messageStringBuilder(
	sFormat := message,
	arg1 := THIS^.AnyToArg(currentValueAsString),
	arg2 := THIS^.AnyToArg(minimumValueAsString)
);

THIS^.assertorContainer.assertor.assert.dateAndTime.simple.dateAndTime.valueIsMin(
	currentValue	:= valueToTest,
	minimumValue	:= minimumValue,
	message			:= ''
);

THIS^.AssertEquals_BOOL(
	Expected 	:= assertionIsWrong,
	Actual 		:= THIS^.assertorContainer.wasAssertionWrong,
	Message 	:= messageStringBuilder.sOut
);
END_METHOD

(*

short summary
==================
This test method tests ``assert.dateAndTime.simple.dateAndTime.valueIsNotEqualTo``
method of CNM_AssertionInterfaces library, 
it provides the possibility to handover test data via parameter 


.. <legal notes>

legal notes
=================
| SPDX-FileCopyrightText: © 2022 ekvip automation GmbH <info@ekvip.de>
| SPDX-License-Identifier: Apache-2.0
| For details check: Apache-2.0_

.. _Apache-2.0: https://www.apache.org/licenses/LICENSE-2.0

.. </legal notes>

parameters
==========

*)

METHOD testValueIsNotEqualTo 
VAR_INPUT
	(* for the test it's the parameter ``currentValue`` *)
	valueToTest		:DT;
	(* for the test it's the parameter ``unexpectedValue`` *)
	unexpectedValue	:DT;
END_VAR
VAR
	(* just the expectation if the assertion to test must be worng or true *)
	assertionIsWrong		:BOOL;
	(* contains the format string for the test message *)
	message					:Tc2_System.T_MaxString;
	(* TwinCAT printf with the test message *)
	messageStringBuilder	:Tc2_Utilities.FB_FormatString;
	(* dt value of ``currentValue`` as string *)
	currentValueAsString	:STRING(22);
	(* dt value of ``unexpectedValue`` as string *)
	unexpectedValueAsString	:STRING(22);
END_VAR
THIS^.assertorContainer.resetAssertor();

assertionIsWrong := (valueToTest = unexpectedValue);
message := SEL(
	assertionIsWrong,
	'currentValue is %s expectedValue is %s assertion must be TRUE', 
	'currentValue is %s expectedValue is %s assertion must be FALSE'
);
currentValueAsString := TO_STRING(valueToTest);
unexpectedValueAsString := TO_STRING(unexpectedValue);

messageStringBuilder(
	sFormat := message,
	arg1 := THIS^.AnyToArg(currentValueAsString),
	arg2 := THIS^.AnyToArg(unexpectedValueAsString)
);

THIS^.assertorContainer.assertor.assert.dateAndTime.simple.dateAndTime.valueIsNotEqualTo(
	currentValue	:= valueToTest,
	unexpectedValue	:= unexpectedValue,
	message			:= ''
);

THIS^.AssertEquals_BOOL(
	Expected 	:= assertionIsWrong,
	Actual 		:= THIS^.assertorContainer.wasAssertionWrong,
	Message 	:= messageStringBuilder.sOut
);
END_METHOD

END_FUNCTION_BLOCK

// ---- AssertionTester/AssertionTests/DateTimeAssertions/classes/DateAssertionTests.TcPOU
(*

short summary
==================
This class tests all methods of DATE assertions
with various combinations of inputs and checks expected 
outputs are satisfied or not

.. <legal notes>

legal notes
=================
| SPDX-FileCopyrightText: © 2022 ekvip automation GmbH <info@ekvip.de>
| SPDX-License-Identifier: Apache-2.0
| For details check: Apache-2.0_

.. _Apache-2.0: https://www.apache.org/licenses/LICENSE-2.0

.. </legal notes>

methods and properties
======================

*)


FUNCTION_BLOCK DateAssertionTests EXTENDS AbstractAssertorTest
VAR
	
END_VAR
VAR CONSTANT
	(* prefix to unify the test names *)
	TEST_NAME_PREFIX		:STRING := 'assert.dateAndTime.simple.dateOnly.';
	(* max value of a DWORD *)
	{attribute 'hide'}
	MAX_DWORD				:DWORD := 16#FFFF_FFFF;
	(* min value of a DWORD *)
	{attribute 'hide'}
	MIN_DWORD				:DWORD := 16#0000_0000;
	(* only the msb is set *)
	{attribute 'hide'}
	MSB_ONLY				:DWORD := 16#8000_0000;
	(* only the msb is set *)
	{attribute 'hide'}
	LSB_ONLY				:DWORD := 16#0000_0001;
	(* all bits set except the msb *)
	{attribute 'hide'}
	WITHOUT_MSB 			:DWORD := 16#7FFF_FFFF;
	(* for every nibble is the msb set only *)
	{attribute 'hide'}
	ALL_NIBBLE_MSB			:DWORD := 16#8888_8888;
	(* for every nibble is the msb unset only *)
	{attribute 'hide'}
	WITHOUT_NIBBLE_MSB		:DWORD := 16#7777_7777;
	(* for every nibble is the lsb set only *)
	{attribute 'hide'}
	ALL_NIBBLE_LSB			:DWORD := 16#1111_1111;
	(* every bit is set except the lsb *)
	{attribute 'hide'}
	LSB_IS_UNSET			:DWORD := 16#FFFF_FFFE;
	(* max vale of date and time *)
	DATE_MAX				:DATE := TO_DATE(MAX_DWORD);
	(* min vale of date and time *)
	DATE_MIN				:DATE := TO_DATE(MIN_DWORD);
	(* only the msb is set *)
	DATE_MSB_ONLY			:DATE := TO_DATE(MSB_ONLY);
	(* all bits set except the msb *)
	DATE_WITHOUT_MSB 		:DATE := TO_DATE(WITHOUT_MSB);
	(* for every nibble is the msb set only *)
	DATE_ALL_NIBBLE_MSB		:DATE := TO_DATE(ALL_NIBBLE_MSB);
	(* for every nibble is the msb unset only *)
	DATE_WITHOUT_NIBBLE_MSB	:DATE := TO_DATE(WITHOUT_NIBBLE_MSB);
	(* for every nibble is the lsb set only *)
	DATE_ALL_NIBBLE_LSB		:DATE := TO_DATE(ALL_NIBBLE_LSB);	
	(* every bit is set except the lsb *)
	DATE_LSB_IS_UNSET		:DATE := TO_DATE(LSB_IS_UNSET);
	(* only the msb is set *)
	DATE_LSB_ONLY			:DATE := TO_DATE(LSB_ONLY);
END_VAR

THIS^.runValueIsEqualToTests();
THIS^.runValueIsGreaterThanTests();
THIS^.runValueIsInRangeOfTests();
THIS^.runValueIsLessThanTests();
THIS^.runValueIsMaxTests();
THIS^.runValueIsMinTests();
THIS^.runValueIsNotEqualToTests();

(*

short summary
==================
This test method is a helper function to create a unified test name

.. <legal notes>

legal notes
=================
| SPDX-FileCopyrightText: © 2022 ekvip automation GmbH <info@ekvip.de>
| SPDX-License-Identifier: Apache-2.0
| For details check: Apache-2.0_

.. _Apache-2.0: https://www.apache.org/licenses/LICENSE-2.0

.. </legal notes>

parameters
==========

*)

METHOD PROTECTED getTestNameFor :Tc2_System.T_MaxString
VAR_INPUT
	(* name of the method to test, to create a unified test name *)
	nameOfMethodToTest	:Tc2_System.T_MaxString;
END_VAR
getTestNameFor := Tc2_Standard.CONCAT(THIS^.TEST_NAME_PREFIX, nameOfMethodToTest);
END_METHOD

(*

short summary
==================
This test method tests ``assert.dateAndTime.simple.dateOnly.valueIsEqualTo``
method of CNM_AssertionInterfaces library with various inputs

.. <legal notes>

legal notes
=================
| SPDX-FileCopyrightText: © 2022 ekvip automation GmbH <info@ekvip.de>
| SPDX-License-Identifier: Apache-2.0
| For details check: Apache-2.0_

.. _Apache-2.0: https://www.apache.org/licenses/LICENSE-2.0

.. </legal notes>

*)

METHOD runValueIsEqualToTests
RETURN (NOT TcUnit.TEST_ORDERED(THIS^.getTestNameFor('valueIsEqualTo')));

THIS^.testValueIsEqualTo(
	valueToTest := THIS^.DATE_MAX,
	expected := THIS^.DATE_MAX
);
THIS^.testValueIsEqualTo(
	valueToTest := THIS^.DATE_MIN,
	expected := THIS^.DATE_MIN
);
THIS^.testValueIsEqualTo(
	valueToTest := THIS^.DATE_MIN,
	expected := THIS^.DATE_MAX
);
THIS^.testValueIsEqualTo(
	valueToTest := THIS^.DATE_MAX,
	expected := THIS^.DATE_MIN
);
THIS^.testValueIsEqualTo(
	valueToTest := THIS^.DATE_ALL_NIBBLE_LSB,
	expected := THIS^.DATE_ALL_NIBBLE_LSB
);
THIS^.testValueIsEqualTo(
	valueToTest := THIS^.DATE_LSB_ONLY,
	expected := THIS^.DATE_MSB_ONLY
);
THIS^.testValueIsEqualTo(
	valueToTest := THIS^.DATE_MSB_ONLY,
	expected := THIS^.DATE_MSB_ONLY
);
THIS^.testValueIsEqualTo(
	valueToTest := THIS^.DATE_MSB_ONLY,
	expected := THIS^.DATE_LSB_ONLY
);

TcUnit.TEST_FINISHED();
END_METHOD

(*

short summary
==================
This test method tests ``assert.dateAndTime.simple.dateOnly.valueIsGreaterThan``
method of CNM_AssertionInterfaces library with various inputs

.. <legal notes>

legal notes
=================
| SPDX-FileCopyrightText: © 2022 ekvip automation GmbH <info@ekvip.de>
| SPDX-License-Identifier: Apache-2.0
| For details check: Apache-2.0_

.. _Apache-2.0: https://www.apache.org/licenses/LICENSE-2.0

.. </legal notes>

*)

METHOD runValueIsGreaterThanTests
RETURN (NOT TcUnit.TEST_ORDERED(THIS^.getTestNameFor('valueIsGreaterThan')));

THIS^.testValueIsGreaterThan(
	valueToTest := THIS^.DATE_MAX,
	lessValue := THIS^.DATE_MAX
);
THIS^.testValueIsGreaterThan(
	valueToTest := THIS^.DATE_MIN,
	lessValue := THIS^.DATE_MIN
);
THIS^.testValueIsGreaterThan(
	valueToTest := THIS^.DATE_MIN,
	lessValue := THIS^.DATE_MAX
);
THIS^.testValueIsGreaterThan(
	valueToTest := THIS^.DATE_MAX,
	lessValue := THIS^.DATE_MIN
);
THIS^.testValueIsGreaterThan(
	valueToTest := THIS^.DATE_ALL_NIBBLE_LSB,
	lessValue := THIS^.DATE_ALL_NIBBLE_LSB
);
THIS^.testValueIsGreaterThan(
	valueToTest := THIS^.DATE_ALL_NIBBLE_MSB,
	lessValue := THIS^.DATE_ALL_NIBBLE_LSB
);
THIS^.testValueIsGreaterThan(
	valueToTest := THIS^.DATE_ALL_NIBBLE_LSB,
	lessValue := THIS^.DATE_ALL_NIBBLE_MSB
);
THIS^.testValueIsGreaterThan(
	valueToTest := THIS^.DATE_LSB_ONLY,
	lessValue := THIS^.DATE_MSB_ONLY
);
THIS^.testValueIsGreaterThan(
	valueToTest := THIS^.DATE_MSB_ONLY,
	lessValue := THIS^.DATE_MSB_ONLY
);
THIS^.testValueIsGreaterThan(
	valueToTest := THIS^.DATE_MSB_ONLY,
	lessValue := THIS^.DATE_LSB_ONLY
);
THIS^.testValueIsGreaterThan(
	valueToTest := THIS^.DATE_LSB_IS_UNSET,
	lessValue := THIS^.DATE_MAX
);
THIS^.testValueIsGreaterThan(
	valueToTest := THIS^.DATE_MAX,
	lessValue := THIS^.DATE_LSB_IS_UNSET
);
TcUnit.TEST_FINISHED();
END_METHOD

(*

short summary
==================
This test method tests ``assert.dateAndTime.simple.dateOnly.valueIsInRangeOf``
method of CNM_AssertionInterfaces library with various inputs

.. <legal notes>

legal notes
=================
| SPDX-FileCopyrightText: © 2022 ekvip automation GmbH <info@ekvip.de>
| SPDX-License-Identifier: Apache-2.0
| For details check: Apache-2.0_

.. _Apache-2.0: https://www.apache.org/licenses/LICENSE-2.0

.. </legal notes>

*)

METHOD runValueIsInRangeOfTests
RETURN (NOT TcUnit.TEST_ORDERED(THIS^.getTestNameFor('valueIsInRangeOf')));

THIS^.testValueIsInRangeOf(
	lowerLimit := THIS^.DATE_MIN,
	valueToTest := THIS^.DATE_MAX,
	upperLimit	:= THIS^.DATE_MAX
);
THIS^.testValueIsInRangeOf(
	lowerLimit := THIS^.DATE_MIN,
	valueToTest := THIS^.DATE_MIN,
	upperLimit	:= THIS^.DATE_MAX
);
THIS^.testValueIsInRangeOf(
	lowerLimit := THIS^.DATE_MAX,
	valueToTest := THIS^.DATE_MAX,
	upperLimit	:= THIS^.DATE_MIN
);
THIS^.testValueIsInRangeOf(
	lowerLimit := THIS^.DATE_MAX,
	valueToTest := THIS^.DATE_MIN,
	upperLimit	:= THIS^.DATE_MIN
);
THIS^.testValueIsInRangeOf(
	lowerLimit := THIS^.DATE_LSB_IS_UNSET,
	valueToTest := THIS^.DATE_MIN,
	upperLimit	:= THIS^.DATE_MAX
);
THIS^.testValueIsInRangeOf(
	lowerLimit := THIS^.DATE_MIN,
	valueToTest := THIS^.DATE_LSB_IS_UNSET,
	upperLimit	:= THIS^.DATE_MAX
);
THIS^.testValueIsInRangeOf(
	lowerLimit := THIS^.DATE_LSB_IS_UNSET,
	valueToTest := THIS^.DATE_LSB_IS_UNSET,
	upperLimit	:= THIS^.DATE_LSB_IS_UNSET
);
THIS^.testValueIsInRangeOf(
	lowerLimit := THIS^.DATE_ALL_NIBBLE_LSB,
	valueToTest := THIS^.DATE_LSB_IS_UNSET,
	upperLimit	:= THIS^.DATE_ALL_NIBBLE_MSB
);
THIS^.testValueIsInRangeOf(
	lowerLimit := THIS^.DATE_LSB_IS_UNSET,
	valueToTest := THIS^.DATE_ALL_NIBBLE_LSB,
	upperLimit	:= THIS^.DATE_ALL_NIBBLE_MSB
);
THIS^.testValueIsInRangeOf(
	lowerLimit := THIS^.DATE_LSB_ONLY,
	valueToTest := THIS^.DATE_WITHOUT_MSB,
	upperLimit	:= THIS^.DATE_MSB_ONLY
);
THIS^.testValueIsInRangeOf(
	lowerLimit := THIS^.DATE_WITHOUT_MSB,
	valueToTest := THIS^.DATE_LSB_ONLY,
	upperLimit	:= THIS^.DATE_MSB_ONLY
);
THIS^.testValueIsInRangeOf(
	lowerLimit := THIS^.DATE_WITHOUT_NIBBLE_MSB,
	valueToTest := THIS^.DATE_MAX,
	upperLimit	:= THIS^.DATE_ALL_NIBBLE_MSB
);
THIS^.testValueIsInRangeOf(
	lowerLimit := THIS^.DATE_WITHOUT_NIBBLE_MSB,
	valueToTest := THIS^.DATE_MIN,
	upperLimit	:= THIS^.DATE_ALL_NIBBLE_MSB
);
THIS^.testValueIsInRangeOf(
	lowerLimit := THIS^.DATE_WITHOUT_NIBBLE_MSB,
	valueToTest := THIS^.DATE_WITHOUT_NIBBLE_MSB,
	upperLimit	:= THIS^.DATE_ALL_NIBBLE_MSB
);
THIS^.testValueIsInRangeOf(
	lowerLimit := THIS^.DATE_WITHOUT_NIBBLE_MSB,
	valueToTest := THIS^.DATE_ALL_NIBBLE_MSB,
	upperLimit	:= THIS^.DATE_ALL_NIBBLE_MSB
);
TcUnit.TEST_FINISHED();
END_METHOD

(*

short summary
==================
This test method tests ``assert.dateAndTime.simple.dateOnly.valueIsLessThan``
method of CNM_AssertionInterfaces library with various inputs

.. <legal notes>

legal notes
=================
| SPDX-FileCopyrightText: © 2022 ekvip automation GmbH <info@ekvip.de>
| SPDX-License-Identifier: Apache-2.0
| For details check: Apache-2.0_

.. _Apache-2.0: https://www.apache.org/licenses/LICENSE-2.0

.. </legal notes>

*)

METHOD runValueIsLessThanTests
RETURN (NOT TcUnit.TEST_ORDERED(THIS^.getTestNameFor('valueIsLessThan')));

THIS^.testValueIsLessThan(
	valueToTest := THIS^.DATE_MAX,
	greaterValue := THIS^.DATE_MAX
);
THIS^.testValueIsLessThan(
	valueToTest := THIS^.DATE_MIN,
	greaterValue := THIS^.DATE_MIN
);
THIS^.testValueIsLessThan(
	valueToTest := THIS^.DATE_MIN,
	greaterValue := THIS^.DATE_MAX
);
THIS^.testValueIsLessThan(
	valueToTest := THIS^.DATE_MAX,
	greaterValue := THIS^.DATE_MIN
);
THIS^.testValueIsLessThan(
	valueToTest := THIS^.DATE_ALL_NIBBLE_LSB,
	greaterValue := THIS^.DATE_ALL_NIBBLE_LSB
);
THIS^.testValueIsLessThan(
	valueToTest := THIS^.DATE_ALL_NIBBLE_MSB,
	greaterValue := THIS^.DATE_ALL_NIBBLE_LSB
);
THIS^.testValueIsLessThan(
	valueToTest := THIS^.DATE_ALL_NIBBLE_LSB,
	greaterValue := THIS^.DATE_ALL_NIBBLE_MSB
);
THIS^.testValueIsLessThan(
	valueToTest := THIS^.DATE_LSB_ONLY,
	greaterValue := THIS^.DATE_MSB_ONLY
);
THIS^.testValueIsLessThan(
	valueToTest := THIS^.DATE_MSB_ONLY,
	greaterValue := THIS^.DATE_MSB_ONLY
);
THIS^.testValueIsLessThan(
	valueToTest := THIS^.DATE_MSB_ONLY,
	greaterValue := THIS^.DATE_LSB_ONLY
);
THIS^.testValueIsLessThan(
	valueToTest := THIS^.DATE_LSB_IS_UNSET,
	greaterValue := THIS^.DATE_MAX
);
THIS^.testValueIsLessThan(
	valueToTest := THIS^.DATE_MAX,
	greaterValue := THIS^.DATE_LSB_IS_UNSET
);
TcUnit.TEST_FINISHED();
END_METHOD

(*

short summary
==================
This test method tests ``assert.dateAndTime.simple.dateOnly.valueIsMax``
method of CNM_AssertionInterfaces library with various inputs

.. <legal notes>

legal notes
=================
| SPDX-FileCopyrightText: © 2022 ekvip automation GmbH <info@ekvip.de>
| SPDX-License-Identifier: Apache-2.0
| For details check: Apache-2.0_

.. _Apache-2.0: https://www.apache.org/licenses/LICENSE-2.0

.. </legal notes>

*)

METHOD runValueIsMaxTests
RETURN (NOT TcUnit.TEST_ORDERED(THIS^.getTestNameFor('valueIsMax')));

THIS^.testValueIsMax(
	valueToTest := THIS^.DATE_MAX,
	maximumValue := THIS^.DATE_MAX
);
THIS^.testValueIsMax(
	valueToTest := THIS^.DATE_MIN,
	maximumValue := THIS^.DATE_MIN
);
THIS^.testValueIsMax(
	valueToTest := THIS^.DATE_MIN,
	maximumValue := THIS^.DATE_MAX
);
THIS^.testValueIsMax(
	valueToTest := THIS^.DATE_MAX,
	maximumValue := THIS^.DATE_MIN
);
THIS^.testValueIsMax(
	valueToTest := THIS^.DATE_ALL_NIBBLE_LSB,
	maximumValue := THIS^.DATE_ALL_NIBBLE_LSB
);
THIS^.testValueIsMax(
	valueToTest := THIS^.DATE_ALL_NIBBLE_MSB,
	maximumValue := THIS^.DATE_ALL_NIBBLE_LSB
);
THIS^.testValueIsMax(
	valueToTest := THIS^.DATE_ALL_NIBBLE_LSB,
	maximumValue := THIS^.DATE_ALL_NIBBLE_MSB
);
THIS^.testValueIsMax(
	valueToTest := THIS^.DATE_LSB_ONLY,
	maximumValue := THIS^.DATE_MSB_ONLY
);
THIS^.testValueIsMax(
	valueToTest := THIS^.DATE_MSB_ONLY,
	maximumValue := THIS^.DATE_MSB_ONLY
);
THIS^.testValueIsMax(
	valueToTest := THIS^.DATE_MSB_ONLY,
	maximumValue := THIS^.DATE_LSB_ONLY
);
THIS^.testValueIsMax(
	valueToTest := THIS^.DATE_LSB_IS_UNSET,
	maximumValue := THIS^.DATE_MAX
);
THIS^.testValueIsMax(
	valueToTest := THIS^.DATE_MAX,
	maximumValue := THIS^.DATE_LSB_IS_UNSET
);
TcUnit.TEST_FINISHED();
END_METHOD

(*

short summary
==================
This test method tests ``assert.dateAndTime.simple.dateOnly.valueIsMin``
method of CNM_AssertionInterfaces library with various inputs

.. <legal notes>

legal notes
=================
| SPDX-FileCopyrightText: © 2022 ekvip automation GmbH <info@ekvip.de>
| SPDX-License-Identifier: Apache-2.0
| For details check: Apache-2.0_

.. _Apache-2.0: https://www.apache.org/licenses/LICENSE-2.0

.. </legal notes>

*)

METHOD runValueIsMinTests
RETURN (NOT TcUnit.TEST_ORDERED(THIS^.getTestNameFor('valueIsMin')));

THIS^.testValueIsMin(
	valueToTest := THIS^.DATE_MAX,
	minimumValue := THIS^.DATE_MAX
);
THIS^.testValueIsMin(
	valueToTest := THIS^.DATE_MIN,
	minimumValue := THIS^.DATE_MIN
);
THIS^.testValueIsMin(
	valueToTest := THIS^.DATE_MIN,
	minimumValue := THIS^.DATE_MAX
);
THIS^.testValueIsMin(
	valueToTest := THIS^.DATE_MAX,
	minimumValue := THIS^.DATE_MIN
);
THIS^.testValueIsMin(
	valueToTest := THIS^.DATE_ALL_NIBBLE_LSB,
	minimumValue := THIS^.DATE_ALL_NIBBLE_LSB
);
THIS^.testValueIsMin(
	valueToTest := THIS^.DATE_ALL_NIBBLE_MSB,
	minimumValue := THIS^.DATE_ALL_NIBBLE_LSB
);
THIS^.testValueIsMin(
	valueToTest := THIS^.DATE_ALL_NIBBLE_LSB,
	minimumValue := THIS^.DATE_ALL_NIBBLE_MSB
);
THIS^.testValueIsMin(
	valueToTest := THIS^.DATE_LSB_ONLY,
	minimumValue := THIS^.DATE_MSB_ONLY
);
THIS^.testValueIsMin(
	valueToTest := THIS^.DATE_MSB_ONLY,
	minimumValue := THIS^.DATE_MSB_ONLY
);
THIS^.testValueIsMin(
	valueToTest := THIS^.DATE_MSB_ONLY,
	minimumValue := THIS^.DATE_LSB_ONLY
);
THIS^.testValueIsMin(
	valueToTest := THIS^.DATE_LSB_IS_UNSET,
	minimumValue := THIS^.DATE_MAX
);
THIS^.testValueIsMin(
	valueToTest := THIS^.DATE_MAX,
	minimumValue := THIS^.DATE_LSB_IS_UNSET
);
TcUnit.TEST_FINISHED();
END_METHOD

(*

short summary
==================
This test method tests ``assert.dateAndTime.simple.dateOnly.valueIsNotEqualTo``
method of CNM_AssertionInterfaces library with various inputs

.. <legal notes>

legal notes
=================
| SPDX-FileCopyrightText: © 2022 ekvip automation GmbH <info@ekvip.de>
| SPDX-License-Identifier: Apache-2.0
| For details check: Apache-2.0_

.. _Apache-2.0: https://www.apache.org/licenses/LICENSE-2.0

.. </legal notes>

*)

METHOD runValueIsNotEqualToTests
RETURN (NOT TcUnit.TEST_ORDERED(THIS^.getTestNameFor('valueIsNotEqualTo')));

THIS^.testValueIsNotEqualTo(
	valueToTest := THIS^.DATE_MAX,
	unexpectedValue := THIS^.DATE_MAX
);
THIS^.testValueIsNotEqualTo(
	valueToTest := THIS^.DATE_MIN,
	unexpectedValue := THIS^.DATE_MIN
);
THIS^.testValueIsNotEqualTo(
	valueToTest := THIS^.DATE_MIN,
	unexpectedValue := THIS^.DATE_MAX
);
THIS^.testValueIsNotEqualTo(
	valueToTest := THIS^.DATE_MAX,
	unexpectedValue := THIS^.DATE_MIN
);
THIS^.testValueIsNotEqualTo(
	valueToTest := THIS^.DATE_ALL_NIBBLE_LSB,
	unexpectedValue := THIS^.DATE_ALL_NIBBLE_LSB
);
THIS^.testValueIsNotEqualTo(
	valueToTest := THIS^.DATE_LSB_ONLY,
	unexpectedValue := THIS^.DATE_MSB_ONLY
);
THIS^.testValueIsNotEqualTo(
	valueToTest := THIS^.DATE_MSB_ONLY,
	unexpectedValue := THIS^.DATE_MSB_ONLY
);
THIS^.testValueIsNotEqualTo(
	valueToTest := THIS^.DATE_MSB_ONLY,
	unexpectedValue := THIS^.DATE_LSB_ONLY
);

TcUnit.TEST_FINISHED();
END_METHOD

(*

short summary
==================
This test method tests ``assert.dateAndTime.simple.dateOnly.valueIsEqualTo``
method of CNM_AssertionInterfaces library, 
it provides the possibility to handover test data via parameter 


.. <legal notes>

legal notes
=================
| SPDX-FileCopyrightText: © 2022 ekvip automation GmbH <info@ekvip.de>
| SPDX-License-Identifier: Apache-2.0
| For details check: Apache-2.0_

.. _Apache-2.0: https://www.apache.org/licenses/LICENSE-2.0

.. </legal notes>

parameters
==========

*)

METHOD testValueIsEqualTo 
VAR_INPUT
	(* for the test it's the parameter ``currentValue`` *)
	valueToTest	:DATE;
	(* for the test it's the parameter ``expectedValue`` *)
	expected	:DATE;
END_VAR
VAR
	(* just the expectation if the assertion to test must be worng or true *)
	assertionIsWrong		:BOOL;
	(* contains the format string for the test message *)
	message					:Tc2_System.T_MaxString;
	(* TwinCAT printf with the test message *)
	messageStringBuilder	:Tc2_Utilities.FB_FormatString;
	(* DATE value of ``currentValue`` as string *)
	currentValueAsString	:STRING(22);
	(* DATE value of ``expectedValue`` as string *)
	expectedValueAsString	:STRING(22);
END_VAR
THIS^.assertorContainer.resetAssertor();

assertionIsWrong := (valueToTest <> expected);
message := SEL(
	assertionIsWrong,
	'currentValue is %s expectedValue is %s assertion must be TRUE', 
	'currentValue is %s expectedValue is %s assertion must be FALSE'
);
currentValueAsString := TO_STRING(valueToTest);
expectedValueAsString := TO_STRING(expected);

messageStringBuilder(
	sFormat := message,
	arg1 := THIS^.AnyToArg(currentValueAsString),
	arg2 := THIS^.AnyToArg(expectedValueAsString)
);

THIS^.assertorContainer.assertor.assert.dateAndTime.simple.dateOnly.valueIsEqualTo(
	currentValue	:= valueToTest,
	expectedValue	:= expected,
	message			:= ''
);

THIS^.AssertEquals_BOOL(
	Expected 	:= assertionIsWrong,
	Actual 		:= THIS^.assertorContainer.wasAssertionWrong,
	Message 	:= messageStringBuilder.sOut
);
END_METHOD

(*

short summary
==================
This test method tests ``assert.dateAndTime.simple.dateOnly.valueIsGreaterThan``
method of CNM_AssertionInterfaces library, 
it provides the possibility to handover test data via parameter 


.. <legal notes>

legal notes
=================
| SPDX-FileCopyrightText: © 2022 ekvip automation GmbH <info@ekvip.de>
| SPDX-License-Identifier: Apache-2.0
| For details check: Apache-2.0_

.. _Apache-2.0: https://www.apache.org/licenses/LICENSE-2.0

.. </legal notes>

parameters
==========

*)

METHOD testValueIsGreaterThan 
VAR_INPUT
	(* for the test it's the parameter ``currentValue`` *)
	valueToTest	:DATE;
	(* for the test it's the parameter ``lessValue`` *)
	lessValue	:DATE;
END_VAR
VAR
	(* just the expectation if the assertion to test must be worng or true *)
	assertionIsWrong		:BOOL;
	(* contains the format string for the test message *)
	message					:Tc2_System.T_MaxString;
	(* TwinCAT printf with the test message *)
	messageStringBuilder	:Tc2_Utilities.FB_FormatString;
	(* DATE value of ``currentValue`` as string *)
	currentValueAsString	:STRING(22);
	(* DATE value of ``lessValue`` as string *)
	lessValueAsString		:STRING(22);
END_VAR
THIS^.assertorContainer.resetAssertor();

assertionIsWrong := (valueToTest <= lessValue);
message := SEL(
	assertionIsWrong,
	'currentValue is %s lessValue is %s assertion must be TRUE', 
	'currentValue is %s lessValue is %s assertion must be FALSE'
);
currentValueAsString := TO_STRING(valueToTest);
lessValueAsString := TO_STRING(lessValue);

messageStringBuilder(
	sFormat := message,
	arg1 := THIS^.AnyToArg(currentValueAsString),
	arg2 := THIS^.AnyToArg(lessValueAsString)
);

THIS^.assertorContainer.assertor.assert.dateAndTime.simple.dateOnly.valueIsGreaterThan(
	currentValue	:= valueToTest,
	lessValue		:= lessValue,
	message			:= ''
);

THIS^.AssertEquals_BOOL(
	Expected 	:= assertionIsWrong,
	Actual 		:= THIS^.assertorContainer.wasAssertionWrong,
	Message 	:= messageStringBuilder.sOut
);
END_METHOD

(*

short summary
==================
This test method tests ``assert.dateAndTime.simple.dateOnly.valueIsInRangeOf``
method of CNM_AssertionInterfaces library, 
it provides the possibility to handover test data via parameter 


.. <legal notes>

legal notes
=================
| SPDX-FileCopyrightText: © 2022 ekvip automation GmbH <info@ekvip.de>
| SPDX-License-Identifier: Apache-2.0
| For details check: Apache-2.0_

.. _Apache-2.0: https://www.apache.org/licenses/LICENSE-2.0

.. </legal notes>

parameters
==========

*)

METHOD testValueIsInRangeOf 
VAR_INPUT
	(* for the test it's the parameter ``lowerLimit`` *)
	lowerLimit	:DATE;
	(* for the test it's the parameter ``currentValue`` *)
	valueToTest	:DATE;
	(* for the test it's the parameter ``upperLimit`` *)
	upperLimit	:DATE;
END_VAR
VAR
	(* just the expectation if the assertion to test must be worng or true *)
	assertionIsWrong		:BOOL;
	(* contains the format string for the test message *)
	message					:Tc2_System.T_MaxString;
	(* TwinCAT printf with the test message *)
	messageStringBuilder	:Tc2_Utilities.FB_FormatString;
	(* DATE value of ``lowerLimit`` as string *)
	lowerLimitAsString		:STRING(22);
	(* DATE value of ``currentValue`` as string *)
	currentValueAsString	:STRING(22);
	(* DATE value of ``upperLimit`` as string *)
	upperLimitAsString		:STRING(22);

END_VAR
THIS^.assertorContainer.resetAssertor();

assertionIsWrong := ((valueToTest < lowerLimit) OR (valueToTest > upperLimit));
message := SEL(
	assertionIsWrong,
	'lowerLimit is %s currentValue is %s upperLimit is %s assertion must be TRUE', 
	'lowerLimit is %s currentValue is %s upperLimit is %s assertion must be FALSE'
);
lowerLimitAsString		:= TO_STRING(lowerLimit);
currentValueAsString	:= TO_STRING(valueToTest);
upperLimitAsString		:= TO_STRING(upperLimit);

messageStringBuilder(
	sFormat := message,
	arg1 := THIS^.AnyToArg(lowerLimitAsString),
	arg2 := THIS^.AnyToArg(currentValueAsString),
	arg3 := THIS^.AnyToArg(upperLimitAsString)
);

THIS^.assertorContainer.assertor.assert.dateAndTime.simple.dateOnly.valueIsInRangeOf(
	lowerLimit		:= lowerLimit,
	currentValue	:= valueToTest,
	upperLimit		:= upperLimit,
	message			:= ''
);

THIS^.AssertEquals_BOOL(
	Expected 	:= assertionIsWrong,
	Actual 		:= THIS^.assertorContainer.wasAssertionWrong,
	Message 	:= messageStringBuilder.sOut
);
END_METHOD

(*

short summary
==================
This test method tests ``assert.dateAndTime.simple.dateOnly.valueIsLessThan``
method of CNM_AssertionInterfaces library, 
it provides the possibility to handover test data via parameter 


.. <legal notes>

legal notes
=================
| SPDX-FileCopyrightText: © 2022 ekvip automation GmbH <info@ekvip.de>
| SPDX-License-Identifier: Apache-2.0
| For details check: Apache-2.0_

.. _Apache-2.0: https://www.apache.org/licenses/LICENSE-2.0

.. </legal notes>

parameters
==========

*)

METHOD testValueIsLessThan 
VAR_INPUT
	(* for the test it's the parameter ``currentValue`` *)
	valueToTest		:DATE;
	(* for the test it's the parameter ``greaterValue`` *)
	greaterValue	:DATE;
END_VAR
VAR
	(* just the expectation if the assertion to test must be worng or true *)
	assertionIsWrong		:BOOL;
	(* contains the format string for the test message *)
	message					:Tc2_System.T_MaxString;
	(* TwinCAT printf with the test message *)
	messageStringBuilder	:Tc2_Utilities.FB_FormatString;
	(* DATE value of ``currentValue`` as string *)
	currentValueAsString	:STRING(22);
	(* DATE value of ``greaterValue`` as string *)
	greaterValueAsString	:STRING(22);
END_VAR
THIS^.assertorContainer.resetAssertor();

assertionIsWrong := (valueToTest >= greaterValue);
message := SEL(
	assertionIsWrong,
	'currentValue is %s greaterValue is %s assertion must be TRUE', 
	'currentValue is %s greaterValue is %s assertion must be FALSE'
);
currentValueAsString := TO_STRING(valueToTest);
greaterValueAsString := TO_STRING(greaterValue);

messageStringBuilder(
	sFormat := message,
	arg1 := THIS^.AnyToArg(currentValueAsString),
	arg2 := THIS^.AnyToArg(greaterValueAsString)
);

THIS^.assertorContainer.assertor.assert.dateAndTime.simple.dateOnly.valueIsLessThan(
	currentValue	:= valueToTest,
	greaterValue	:= greaterValue,
	message			:= ''
);

THIS^.AssertEquals_BOOL(
	Expected 	:= assertionIsWrong,
	Actual 		:= THIS^.assertorContainer.wasAssertionWrong,
	Message 	:= messageStringBuilder.sOut
);
END_METHOD

(*

short summary
==================
This test method tests ``assert.dateAndTime.simple.dateOnly.valueIsMax``
method of CNM_AssertionInterfaces library, 
it provides the possibility to handover test data via parameter 


.. <legal notes>

legal notes
=================
| SPDX-FileCopyrightText: © 2022 ekvip automation GmbH <info@ekvip.de>
| SPDX-License-Identifier: Apache-2.0
| For details check: Apache-2.0_

.. _Apache-2.0: https://www.apache.org/licenses/LICENSE-2.0

.. </legal notes>

parameters
==========

*)

METHOD testValueIsMax 
VAR_INPUT
	(* for the test it's the parameter ``currentValue`` *)
	valueToTest		:DATE;
	(* for the test it's the parameter ``greaterValue`` *)
	maximumValue	:DATE;
END_VAR
VAR
	(* just the expectation if the assertion to test must be worng or true *)
	assertionIsWrong		:BOOL;
	(* contains the format string for the test message *)
	message					:Tc2_System.T_MaxString;
	(* TwinCAT printf with the test message *)
	messageStringBuilder	:Tc2_Utilities.FB_FormatString;
	(* DATE value of ``currentValue`` as string *)
	currentValueAsString	:STRING(22);
	(* DATE value of ``maximumValue`` as string *)
	maximumValueAsString	:STRING(22);
END_VAR
THIS^.assertorContainer.resetAssertor();

assertionIsWrong := (valueToTest > maximumValue);
message := SEL(
	assertionIsWrong,
	'currentValue is %s maximumValue is %s assertion must be TRUE', 
	'currentValue is %s maximumValue is %s assertion must be FALSE'
);
currentValueAsString := TO_STRING(valueToTest);
maximumValueAsString := TO_STRING(maximumValue);

messageStringBuilder(
	sFormat := message,
	arg1 := THIS^.AnyToArg(currentValueAsString),
	arg2 := THIS^.AnyToArg(maximumValueAsString)
);

THIS^.assertorContainer.assertor.assert.dateAndTime.simple.dateOnly.valueIsMax(
	currentValue	:= valueToTest,
	maximumValue	:= maximumValue,
	message			:= ''
);

THIS^.AssertEquals_BOOL(
	Expected 	:= assertionIsWrong,
	Actual 		:= THIS^.assertorContainer.wasAssertionWrong,
	Message 	:= messageStringBuilder.sOut
);
END_METHOD

(*

short summary
==================
This test method tests ``assert.dateAndTime.simple.dateOnly.valueIsMin``
method of CNM_AssertionInterfaces library, 
it provides the possibility to handover test data via parameter 


.. <legal notes>

legal notes
=================
| SPDX-FileCopyrightText: © 2022 ekvip automation GmbH <info@ekvip.de>
| SPDX-License-Identifier: Apache-2.0
| For details check: Apache-2.0_

.. _Apache-2.0: https://www.apache.org/licenses/LICENSE-2.0

.. </legal notes>

parameters
==========

*)

METHOD testValueIsMin 
VAR_INPUT
	(* for the test it's the parameter ``currentValue`` *)
	valueToTest		:DATE;
	(* for the test it's the parameter ``greaterValue`` *)
	minimumValue	:DATE;
END_VAR
VAR
	(* just the expectation if the assertion to test must be worng or true *)
	assertionIsWrong		:BOOL;
	(* contains the format string for the test message *)
	message					:Tc2_System.T_MaxString;
	(* TwinCAT printf with the test message *)
	messageStringBuilder	:Tc2_Utilities.FB_FormatString;
	(* DATE value of ``currentValue`` as string *)
	currentValueAsString	:STRING(22);
	(* DATE value of ``minimumValue`` as string *)
	minimumValueAsString	:STRING(22);
END_VAR
THIS^.assertorContainer.resetAssertor();

assertionIsWrong := (valueToTest < minimumValue);
message := SEL(
	assertionIsWrong,
	'currentValue is %s minimumValue is %s assertion must be TRUE', 
	'currentValue is %s minimumValue is %s assertion must be FALSE'
);
currentValueAsString := TO_STRING(valueToTest);
minimumValueAsString := TO_STRING(minimumValue);

messageStringBuilder(
	sFormat := message,
	arg1 := THIS^.AnyToArg(currentValueAsString),
	arg2 := THIS^.AnyToArg(minimumValueAsString)
);

THIS^.assertorContainer.assertor.assert.dateAndTime.simple.dateOnly.valueIsMin(
	currentValue	:= valueToTest,
	minimumValue	:= minimumValue,
	message			:= ''
);

THIS^.AssertEquals_BOOL(
	Expected 	:= assertionIsWrong,
	Actual 		:= THIS^.assertorContainer.wasAssertionWrong,
	Message 	:= messageStringBuilder.sOut
);
END_METHOD

(*

short summary
==================
This test method tests ``assert.dateAndTime.simple.dateOnly.valueIsNotEqualTo``
method of CNM_AssertionInterfaces library, 
it provides the possibility to handover test data via parameter 


.. <legal notes>

legal notes
=================
| SPDX-FileCopyrightText: © 2022 ekvip automation GmbH <info@ekvip.de>
| SPDX-License-Identifier: Apache-2.0
| For details check: Apache-2.0_

.. _Apache-2.0: https://www.apache.org/licenses/LICENSE-2.0

.. </legal notes>

parameters
==========

*)

METHOD testValueIsNotEqualTo 
VAR_INPUT
	(* for the test it's the parameter ``currentValue`` *)
	valueToTest		:DATE;
	(* for the test it's the parameter ``unexpectedValue`` *)
	unexpectedValue	:DATE;
END_VAR
VAR
	(* just the expectation if the assertion to test must be worng or true *)
	assertionIsWrong		:BOOL;
	(* contains the format string for the test message *)
	message					:Tc2_System.T_MaxString;
	(* TwinCAT printf with the test message *)
	messageStringBuilder	:Tc2_Utilities.FB_FormatString;
	(* DATE value of ``currentValue`` as string *)
	currentValueAsString	:STRING(22);
	(* DATE value of ``unexpectedValue`` as string *)
	unexpectedValueAsString	:STRING(22);
END_VAR
THIS^.assertorContainer.resetAssertor();

assertionIsWrong := (valueToTest = unexpectedValue);
message := SEL(
	assertionIsWrong,
	'currentValue is %s expectedValue is %s assertion must be TRUE', 
	'currentValue is %s expectedValue is %s assertion must be FALSE'
);
currentValueAsString := TO_STRING(valueToTest);
unexpectedValueAsString := TO_STRING(unexpectedValue);

messageStringBuilder(
	sFormat := message,
	arg1 := THIS^.AnyToArg(currentValueAsString),
	arg2 := THIS^.AnyToArg(unexpectedValueAsString)
);

THIS^.assertorContainer.assertor.assert.dateAndTime.simple.dateOnly.valueIsNotEqualTo(
	currentValue	:= valueToTest,
	unexpectedValue	:= unexpectedValue,
	message			:= ''
);

THIS^.AssertEquals_BOOL(
	Expected 	:= assertionIsWrong,
	Actual 		:= THIS^.assertorContainer.wasAssertionWrong,
	Message 	:= messageStringBuilder.sOut
);
END_METHOD

END_FUNCTION_BLOCK

// ---- AssertionTester/AssertionTests/DateTimeAssertions/classes/LDateAssertionTests.TcPOU
FUNCTION_BLOCK LDateAssertionTests EXTENDS AbstractAssertorTest

VAR
	
END_VAR

VAR CONSTANT
	(* prefix to unify the test names *)
	TEST_NAME_PREFIX			:STRING := 'assert.dateAndTime.long.dateOnly.';
	(* max value of a LWORD *)
	{attribute 'hide'}
	MAX_LWORD					:LWORD := 16#FFFF_FFFF_FFFF_FFFF;
	(* min value of a LWORD *)
	{attribute 'hide'}
	MIN_LWORD					:LWORD := 16#0000_0000_0000_0000;
	(* only the msb is set *)
	{attribute 'hide'}
	MSB_ONLY					:LWORD := 16#8000_0000_0000_0000;
	(* only the msb is set *)
	{attribute 'hide'}
	LSB_ONLY					:LWORD := 16#0000_0000_0000_0001;
	(* all bits set except the msb *)
	{attribute 'hide'}
	WITHOUT_MSB 				:LWORD := 16#7FFF_FFFF_FFFF_FFFF;
	(* for every nibble is the msb set only *)
	{attribute 'hide'}
	ALL_NIBBLE_MSB				:LWORD := 16#8888_8888_8888_8888;
	(* for every nibble is the msb unset only *)
	{attribute 'hide'}
	WITHOUT_NIBBLE_MSB			:LWORD := 16#7777_7777_7777_7777;
	(* for every nibble is the lsb set only *)
	{attribute 'hide'}
	ALL_NIBBLE_LSB				:LWORD := 16#1111_1111_111_111;
	(* every bit is set except the lsb *)
	{attribute 'hide'}
	LSB_IS_UNSET				:LWORD := 16#FFFF_FFFE_FFFF_FFFF;
	(* max vale of date and time *)
	LDATE_MAX					:LDATE := TO_LDATE(MAX_LWORD);
	(* min vale of date and time *)
	LDATE_MIN					:LDATE := TO_LDATE(MIN_LWORD);
	(* only the msb is set *)
	LDATE_MSB_ONLY				:LDATE := TO_LDATE(MSB_ONLY);
	(* all bits set except the msb *)
	LDATE_WITHOUT_MSB 			:LDATE := TO_LDATE(WITHOUT_MSB);
	(* for every nibble is the msb set only *)
	LDATE_ALL_NIBBLE_MSB		:LDATE := TO_LDATE(ALL_NIBBLE_MSB);
	(* for every nibble is the msb unset only *)
	LDATE_WITHOUT_NIBBLE_MSB	:LDATE := TO_LDATE(WITHOUT_NIBBLE_MSB);
	(* for every nibble is the lsb set only *)
	LDATE_ALL_NIBBLE_LSB		:LDATE := TO_LDATE(ALL_NIBBLE_LSB);	
	(* every bit is set except the lsb *)
	LDATE_LSB_IS_UNSET			:LDATE := TO_LDATE(LSB_IS_UNSET);
	(* only the msb is set *)
	LDATE_LSB_ONLY				:LDATE := TO_LDATE(LSB_ONLY);
END_VAR

THIS^.runValueIsEqualToTests();
THIS^.runValueIsGreaterThanTests();
THIS^.runValueIsInRangeOfTests();
THIS^.runValueIsLessThanTests();
THIS^.runValueIsMaxTests();
THIS^.runValueIsMinTests();
THIS^.runValueIsNotEqualToTests();

METHOD getTestNameFor : Tc2_System.t_MaxString

VAR_INPUT
	(* name of the method to test, to create a unified test name *)
	nameOfMethodToTest	:Tc2_System.T_MaxString;
END_VAR
getTestNameFor := Tc2_Standard.CONCAT(THIS^.TEST_NAME_PREFIX, nameOfMethodToTest);
END_METHOD

(*

short summary
==================
This test method tests ``assert.dateAndTime.long.dateOnly.valueIsEqualTo``
method of CNM_AssertionInterfaces library with various inputs

.. <legal notes>

legal notes
=================
| SPDX-FileCopyrightText: © 2022 ekvip automation GmbH <info@ekvip.de>
| SPDX-License-Identifier: Apache-2.0
| For details check: Apache-2.0_

.. _Apache-2.0: https://www.apache.org/licenses/LICENSE-2.0

.. </legal notes>

*)
METHOD runValueIsEqualToTests
RETURN (NOT TcUnit.TEST_ORDERED(THIS^.getTestNameFor('valueIsEqualTo')));

THIS^.testValueIsEqualTo(
	valueToTest := THIS^.LDATE_MAX,
	expected := THIS^.LDATE_MAX
);
THIS^.testValueIsEqualTo(
	valueToTest := THIS^.LDATE_MIN,
	expected := THIS^.LDATE_MIN
);
THIS^.testValueIsEqualTo(
	valueToTest := THIS^.LDATE_MIN,
	expected := THIS^.LDATE_MAX
);
THIS^.testValueIsEqualTo(
	valueToTest := THIS^.LDATE_MAX,
	expected := THIS^.LDATE_MIN
);
THIS^.testValueIsEqualTo(
	valueToTest := THIS^.LDATE_ALL_NIBBLE_LSB,
	expected := THIS^.LDATE_ALL_NIBBLE_LSB
);
THIS^.testValueIsEqualTo(
	valueToTest := THIS^.LDATE_LSB_ONLY,
	expected := THIS^.LDATE_MSB_ONLY
);
THIS^.testValueIsEqualTo(
	valueToTest := THIS^.LDATE_MSB_ONLY,
	expected := THIS^.LDATE_MSB_ONLY
);
THIS^.testValueIsEqualTo(
	valueToTest := THIS^.LDATE_MSB_ONLY,
	expected := THIS^.LDATE_LSB_ONLY
);

TcUnit.TEST_FINISHED();
END_METHOD

(*

short summary
==================
This test method tests ``assert.dateAndTime.long.dateOnly.valueIsGreaterThan``
method of CNM_AssertionInterfaces library with various inputs

.. <legal notes>

legal notes
=================
| SPDX-FileCopyrightText: © 2022 ekvip automation GmbH <info@ekvip.de>
| SPDX-License-Identifier: Apache-2.0
| For details check: Apache-2.0_

.. _Apache-2.0: https://www.apache.org/licenses/LICENSE-2.0

.. </legal notes>

*)

METHOD runValueIsGreaterThanTests
RETURN (NOT TcUnit.TEST_ORDERED(THIS^.getTestNameFor('valueIsGreaterThan')));

THIS^.testValueIsGreaterThan(
	valueToTest := THIS^.LDATE_MAX,
	lessValue := THIS^.LDATE_MAX
);
THIS^.testValueIsGreaterThan(
	valueToTest := THIS^.LDATE_MIN,
	lessValue := THIS^.LDATE_MIN
);
THIS^.testValueIsGreaterThan(
	valueToTest := THIS^.LDATE_MIN,
	lessValue := THIS^.LDATE_MAX
);
THIS^.testValueIsGreaterThan(
	valueToTest := THIS^.LDATE_MAX,
	lessValue := THIS^.LDATE_MIN
);
THIS^.testValueIsGreaterThan(
	valueToTest := THIS^.LDATE_ALL_NIBBLE_LSB,
	lessValue := THIS^.LDATE_ALL_NIBBLE_LSB
);
THIS^.testValueIsGreaterThan(
	valueToTest := THIS^.LDATE_ALL_NIBBLE_MSB,
	lessValue := THIS^.LDATE_ALL_NIBBLE_LSB
);
THIS^.testValueIsGreaterThan(
	valueToTest := THIS^.LDATE_ALL_NIBBLE_LSB,
	lessValue := THIS^.LDATE_ALL_NIBBLE_MSB
);
THIS^.testValueIsGreaterThan(
	valueToTest := THIS^.LDATE_LSB_ONLY,
	lessValue := THIS^.LDATE_MSB_ONLY
);
THIS^.testValueIsGreaterThan(
	valueToTest := THIS^.LDATE_MSB_ONLY,
	lessValue := THIS^.LDATE_MSB_ONLY
);
THIS^.testValueIsGreaterThan(
	valueToTest := THIS^.LDATE_MSB_ONLY,
	lessValue := THIS^.LDATE_LSB_ONLY
);
THIS^.testValueIsGreaterThan(
	valueToTest := THIS^.LDATE_LSB_IS_UNSET,
	lessValue := THIS^.LDATE_MAX
);
THIS^.testValueIsGreaterThan(
	valueToTest := THIS^.LDATE_MAX,
	lessValue := THIS^.LDATE_LSB_IS_UNSET
);

TcUnit.TEST_FINISHED();
END_METHOD

(*

short summary
==================
This test method tests ``assert.dateAndTime.long.dateOnly.valueIsInRangeOf``
method of CNM_AssertionInterfaces library with various inputs

.. <legal notes>

legal notes
=================
| SPDX-FileCopyrightText: © 2022 ekvip automation GmbH <info@ekvip.de>
| SPDX-License-Identifier: Apache-2.0
| For details check: Apache-2.0_

.. _Apache-2.0: https://www.apache.org/licenses/LICENSE-2.0

.. </legal notes>

*)

METHOD runValueIsInRangeOfTests
RETURN (NOT TcUnit.TEST_ORDERED(THIS^.getTestNameFor('valueIsInRangeOf')));

THIS^.testValueIsInRangeOf(
	lowerLimit := THIS^.LDATE_MIN,
	valueToTest := THIS^.LDATE_MAX,
	upperLimit	:= THIS^.LDATE_MAX
);
THIS^.testValueIsInRangeOf(
	lowerLimit := THIS^.LDATE_MIN,
	valueToTest := THIS^.LDATE_MIN,
	upperLimit	:= THIS^.LDATE_MAX
);
THIS^.testValueIsInRangeOf(
	lowerLimit := THIS^.LDATE_MAX,
	valueToTest := THIS^.LDATE_MAX,
	upperLimit	:= THIS^.LDATE_MIN
);
THIS^.testValueIsInRangeOf(
	lowerLimit := THIS^.LDATE_MAX,
	valueToTest := THIS^.LDATE_MIN,
	upperLimit	:= THIS^.LDATE_MIN
);
THIS^.testValueIsInRangeOf(
	lowerLimit := THIS^.LDATE_LSB_IS_UNSET,
	valueToTest := THIS^.LDATE_MIN,
	upperLimit	:= THIS^.LDATE_MAX
);
THIS^.testValueIsInRangeOf(
	lowerLimit := THIS^.LDATE_MIN,
	valueToTest := THIS^.LDATE_LSB_IS_UNSET,
	upperLimit	:= THIS^.LDATE_MAX
);
THIS^.testValueIsInRangeOf(
	lowerLimit := THIS^.LDATE_LSB_IS_UNSET,
	valueToTest := THIS^.LDATE_LSB_IS_UNSET,
	upperLimit	:= THIS^.LDATE_LSB_IS_UNSET
);
THIS^.testValueIsInRangeOf(
	lowerLimit := THIS^.LDATE_ALL_NIBBLE_LSB,
	valueToTest := THIS^.LDATE_LSB_IS_UNSET,
	upperLimit	:= THIS^.LDATE_ALL_NIBBLE_MSB
);
THIS^.testValueIsInRangeOf(
	lowerLimit := THIS^.LDATE_LSB_IS_UNSET,
	valueToTest := THIS^.LDATE_ALL_NIBBLE_LSB,
	upperLimit	:= THIS^.LDATE_ALL_NIBBLE_MSB
);
THIS^.testValueIsInRangeOf(
	lowerLimit := THIS^.LDATE_LSB_ONLY,
	valueToTest := THIS^.LDATE_WITHOUT_MSB,
	upperLimit	:= THIS^.LDATE_MSB_ONLY
);
THIS^.testValueIsInRangeOf(
	lowerLimit := THIS^.LDATE_WITHOUT_MSB,
	valueToTest := THIS^.LDATE_LSB_ONLY,
	upperLimit	:= THIS^.LDATE_MSB_ONLY
);
THIS^.testValueIsInRangeOf(
	lowerLimit := THIS^.LDATE_WITHOUT_NIBBLE_MSB,
	valueToTest := THIS^.LDATE_MAX,
	upperLimit	:= THIS^.LDATE_ALL_NIBBLE_MSB
);
THIS^.testValueIsInRangeOf(
	lowerLimit := THIS^.LDATE_WITHOUT_NIBBLE_MSB,
	valueToTest := THIS^.LDATE_MIN,
	upperLimit	:= THIS^.LDATE_ALL_NIBBLE_MSB
);
THIS^.testValueIsInRangeOf(
	lowerLimit := THIS^.LDATE_WITHOUT_NIBBLE_MSB,
	valueToTest := THIS^.LDATE_WITHOUT_NIBBLE_MSB,
	upperLimit	:= THIS^.LDATE_ALL_NIBBLE_MSB
);
THIS^.testValueIsInRangeOf(
	lowerLimit := THIS^.LDATE_WITHOUT_NIBBLE_MSB,
	valueToTest := THIS^.LDATE_ALL_NIBBLE_MSB,
	upperLimit	:= THIS^.LDATE_ALL_NIBBLE_MSB
);

TcUnit.TEST_FINISHED();
END_METHOD

(*

short summary
==================
This test method tests ``assert.dateAndTime.long.dateOnly.valueIsLessThan``
method of CNM_AssertionInterfaces library with various inputs

.. <legal notes>

legal notes
=================
| SPDX-FileCopyrightText: © 2022 ekvip automation GmbH <info@ekvip.de>
| SPDX-License-Identifier: Apache-2.0
| For details check: Apache-2.0_

.. _Apache-2.0: https://www.apache.org/licenses/LICENSE-2.0

.. </legal notes>

*)

METHOD runValueIsLessThanTests
RETURN (NOT TcUnit.TEST_ORDERED(THIS^.getTestNameFor('valueIsLessThan')));

THIS^.testValueIsLessThan(
	valueToTest := THIS^.LDATE_MAX,
	greaterValue := THIS^.LDATE_MAX
);
THIS^.testValueIsLessThan(
	valueToTest := THIS^.LDATE_MIN,
	greaterValue := THIS^.LDATE_MIN
);
THIS^.testValueIsLessThan(
	valueToTest := THIS^.LDATE_MIN,
	greaterValue := THIS^.LDATE_MAX
);
THIS^.testValueIsLessThan(
	valueToTest := THIS^.LDATE_MAX,
	greaterValue := THIS^.LDATE_MIN
);
THIS^.testValueIsLessThan(
	valueToTest := THIS^.LDATE_ALL_NIBBLE_LSB,
	greaterValue := THIS^.LDATE_ALL_NIBBLE_LSB
);
THIS^.testValueIsLessThan(
	valueToTest := THIS^.LDATE_ALL_NIBBLE_MSB,
	greaterValue := THIS^.LDATE_ALL_NIBBLE_LSB
);
THIS^.testValueIsLessThan(
	valueToTest := THIS^.LDATE_ALL_NIBBLE_LSB,
	greaterValue := THIS^.LDATE_ALL_NIBBLE_MSB
);
THIS^.testValueIsLessThan(
	valueToTest := THIS^.LDATE_LSB_ONLY,
	greaterValue := THIS^.LDATE_MSB_ONLY
);
THIS^.testValueIsLessThan(
	valueToTest := THIS^.LDATE_MSB_ONLY,
	greaterValue := THIS^.LDATE_MSB_ONLY
);
THIS^.testValueIsLessThan(
	valueToTest := THIS^.LDATE_MSB_ONLY,
	greaterValue := THIS^.LDATE_LSB_ONLY
);
THIS^.testValueIsLessThan(
	valueToTest := THIS^.LDATE_LSB_IS_UNSET,
	greaterValue := THIS^.LDATE_MAX
);
THIS^.testValueIsLessThan(
	valueToTest := THIS^.LDATE_MAX,
	greaterValue := THIS^.LDATE_LSB_IS_UNSET
);

TcUnit.TEST_FINISHED();
END_METHOD

(*

short summary
==================
This test method tests ``assert.dateAndTime.long.dateOnly.valueIsMax``
method of CNM_AssertionInterfaces library with various inputs

.. <legal notes>

legal notes
=================
| SPDX-FileCopyrightText: © 2022 ekvip automation GmbH <info@ekvip.de>
| SPDX-License-Identifier: Apache-2.0
| For details check: Apache-2.0_

.. _Apache-2.0: https://www.apache.org/licenses/LICENSE-2.0

.. </legal notes>

*)

METHOD runValueIsMaxTests
RETURN (NOT TcUnit.TEST_ORDERED(THIS^.getTestNameFor('valueIsMax')));

THIS^.testValueIsMax(
	valueToTest := THIS^.LDATE_MAX,
	maximumValue := THIS^.LDATE_MAX
);
THIS^.testValueIsMax(
	valueToTest := THIS^.LDATE_MIN,
	maximumValue := THIS^.LDATE_MIN
);
THIS^.testValueIsMax(
	valueToTest := THIS^.LDATE_MIN,
	maximumValue := THIS^.LDATE_MAX
);
THIS^.testValueIsMax(
	valueToTest := THIS^.LDATE_MAX,
	maximumValue := THIS^.LDATE_MIN
);
THIS^.testValueIsMax(
	valueToTest := THIS^.LDATE_ALL_NIBBLE_LSB,
	maximumValue := THIS^.LDATE_ALL_NIBBLE_LSB
);
THIS^.testValueIsMax(
	valueToTest := THIS^.LDATE_ALL_NIBBLE_MSB,
	maximumValue := THIS^.LDATE_ALL_NIBBLE_LSB
);
THIS^.testValueIsMax(
	valueToTest := THIS^.LDATE_ALL_NIBBLE_LSB,
	maximumValue := THIS^.LDATE_ALL_NIBBLE_MSB
);
THIS^.testValueIsMax(
	valueToTest := THIS^.LDATE_LSB_ONLY,
	maximumValue := THIS^.LDATE_MSB_ONLY
);
THIS^.testValueIsMax(
	valueToTest := THIS^.LDATE_MSB_ONLY,
	maximumValue := THIS^.LDATE_MSB_ONLY
);
THIS^.testValueIsMax(
	valueToTest := THIS^.LDATE_MSB_ONLY,
	maximumValue := THIS^.LDATE_LSB_ONLY
);
THIS^.testValueIsMax(
	valueToTest := THIS^.LDATE_LSB_IS_UNSET,
	maximumValue := THIS^.LDATE_MAX
);
THIS^.testValueIsMax(
	valueToTest := THIS^.LDATE_MAX,
	maximumValue := THIS^.LDATE_LSB_IS_UNSET
);

TcUnit.TEST_FINISHED();
END_METHOD

(*

short summary
==================
This test method tests ``assert.dateAndTime.long.dateOnly.valueIsMin``
method of CNM_AssertionInterfaces library with various inputs

.. <legal notes>

legal notes
=================
| SPDX-FileCopyrightText: © 2022 ekvip automation GmbH <info@ekvip.de>
| SPDX-License-Identifier: Apache-2.0
| For details check: Apache-2.0_

.. _Apache-2.0: https://www.apache.org/licenses/LICENSE-2.0

.. </legal notes>

*)

METHOD runValueIsMinTests
RETURN (NOT TcUnit.TEST_ORDERED(THIS^.getTestNameFor('valueIsMin')));

THIS^.testValueIsMin(
	valueToTest := THIS^.LDATE_MAX,
	minimumValue := THIS^.LDATE_MAX
);
THIS^.testValueIsMin(
	valueToTest := THIS^.LDATE_MIN,
	minimumValue := THIS^.LDATE_MIN
);
THIS^.testValueIsMin(
	valueToTest := THIS^.LDATE_MIN,
	minimumValue := THIS^.LDATE_MAX
);
THIS^.testValueIsMin(
	valueToTest := THIS^.LDATE_MAX,
	minimumValue := THIS^.LDATE_MIN
);
THIS^.testValueIsMin(
	valueToTest := THIS^.LDATE_ALL_NIBBLE_LSB,
	minimumValue := THIS^.LDATE_ALL_NIBBLE_LSB
);
THIS^.testValueIsMin(
	valueToTest := THIS^.LDATE_ALL_NIBBLE_MSB,
	minimumValue := THIS^.LDATE_ALL_NIBBLE_LSB
);
THIS^.testValueIsMin(
	valueToTest := THIS^.LDATE_ALL_NIBBLE_LSB,
	minimumValue := THIS^.LDATE_ALL_NIBBLE_MSB
);
THIS^.testValueIsMin(
	valueToTest := THIS^.LDATE_LSB_ONLY,
	minimumValue := THIS^.LDATE_MSB_ONLY
);
THIS^.testValueIsMin(
	valueToTest := THIS^.LDATE_MSB_ONLY,
	minimumValue := THIS^.LDATE_MSB_ONLY
);
THIS^.testValueIsMin(
	valueToTest := THIS^.LDATE_MSB_ONLY,
	minimumValue := THIS^.LDATE_LSB_ONLY
);
THIS^.testValueIsMin(
	valueToTest := THIS^.LDATE_LSB_IS_UNSET,
	minimumValue := THIS^.LDATE_MAX
);
THIS^.testValueIsMin(
	valueToTest := THIS^.LDATE_MAX,
	minimumValue := THIS^.LDATE_LSB_IS_UNSET
);

TcUnit.TEST_FINISHED();
END_METHOD

(*

short summary
==================
This test method tests ``assert.dateAndTime.long.dateOnly.valueIsNotEqualTo``
method of CNM_AssertionInterfaces library with various inputs

.. <legal notes>

legal notes
=================
| SPDX-FileCopyrightText: © 2022 ekvip automation GmbH <info@ekvip.de>
| SPDX-License-Identifier: Apache-2.0
| For details check: Apache-2.0_

.. _Apache-2.0: https://www.apache.org/licenses/LICENSE-2.0

.. </legal notes>

*)

METHOD runValueIsNotEqualToTests
RETURN (NOT TcUnit.TEST_ORDERED(THIS^.getTestNameFor('valueIsNotEqualTo')));

THIS^.testValueIsNotEqualTo(
	valueToTest := THIS^.LDATE_MAX,
	unexpectedValue := THIS^.LDATE_MAX
);
THIS^.testValueIsNotEqualTo(
	valueToTest := THIS^.LDATE_MIN,
	unexpectedValue := THIS^.LDATE_MIN
);
THIS^.testValueIsNotEqualTo(
	valueToTest := THIS^.LDATE_MIN,
	unexpectedValue := THIS^.LDATE_MAX
);
THIS^.testValueIsNotEqualTo(
	valueToTest := THIS^.LDATE_MAX,
	unexpectedValue := THIS^.LDATE_MIN
);
THIS^.testValueIsNotEqualTo(
	valueToTest := THIS^.LDATE_ALL_NIBBLE_LSB,
	unexpectedValue := THIS^.LDATE_ALL_NIBBLE_LSB
);
THIS^.testValueIsNotEqualTo(
	valueToTest := THIS^.LDATE_LSB_ONLY,
	unexpectedValue := THIS^.LDATE_MSB_ONLY
);
THIS^.testValueIsNotEqualTo(
	valueToTest := THIS^.LDATE_MSB_ONLY,
	unexpectedValue := THIS^.LDATE_MSB_ONLY
);
THIS^.testValueIsNotEqualTo(
	valueToTest := THIS^.LDATE_MSB_ONLY,
	unexpectedValue := THIS^.LDATE_LSB_ONLY
);

TcUnit.TEST_FINISHED();
END_METHOD


(*

short summary
==================
This test method tests ``assert.dateAndTime.long.dateOnly.valueIsEqualTo``
method of CNM_AssertionInterfaces library, 
it provides the possibility to handover test data via parameter 


.. <legal notes>

legal notes
=================
| SPDX-FileCopyrightText: © 2022 ekvip automation GmbH <info@ekvip.de>
| SPDX-License-Identifier: Apache-2.0
| For details check: Apache-2.0_

.. _Apache-2.0: https://www.apache.org/licenses/LICENSE-2.0

.. </legal notes>

parameters
==========

*)
METHOD testValueIsEqualTo
VAR_INPUT
	(* for the test it's the parameter ``currentValue`` *)
	valueToTest	:LDATE;
	(* for the test it's the parameter ``expectedValue`` *)
	expected	:LDATE;
END_VAR
VAR
	(* just the expectation if the assertion to test must be worng or true *)
	assertionIsWrong		:BOOL;
	(* contains the format string for the test message *)
	message					:Tc2_System.T_MaxString;
	(* TwinCAT printf with the test message *)
	messageStringBuilder	:Tc2_Utilities.FB_FormatString;
	(* LDATE value of ``currentValue`` as string *)
	currentValueAsString	:STRING(22);
	(* LDATE value of ``expectedValue`` as string *)
	expectedValueAsString	:STRING(22);
END_VAR
THIS^.assertorContainer.resetAssertor();

assertionIsWrong := (valueToTest <> expected);

message := SEL(
	assertionIsWrong,
	'currentValue is %s expectedValue is %s assertion must be TRUE', 
	'currentValue is %s expectedValue is %s assertion must be FALSE'
);
currentValueAsString := TO_STRING(valueToTest);
expectedValueAsString := TO_STRING(expected);

messageStringBuilder(
	sFormat := message,
	arg1 := THIS^.AnyToArg(currentValueAsString),
	arg2 := THIS^.AnyToArg(expectedValueAsString)
);

THIS^.assertorContainer.assertor.assert.dateAndTime.long.dateOnly.valueIsEqualTo(
	currentValue	:= valueToTest,
	expectedValue	:= expected,
	message			:= ''
);

THIS^.AssertEquals_BOOL(
	Expected 	:= assertionIsWrong,
	Actual 		:= THIS^.assertorContainer.wasAssertionWrong,
	Message 	:= messageStringBuilder.sOut
);
END_METHOD

(*

short summary
==================
This test method tests ``assert.dateAndTime.long.dateOnly.valueIsGreaterThan``
method of CNM_AssertionInterfaces library, 
it provides the possibility to handover test data via parameter 


.. <legal notes>

legal notes
=================
| SPDX-FileCopyrightText: © 2022 ekvip automation GmbH <info@ekvip.de>
| SPDX-License-Identifier: Apache-2.0
| For details check: Apache-2.0_

.. _Apache-2.0: https://www.apache.org/licenses/LICENSE-2.0

.. </legal notes>

parameters
==========

*)

METHOD testValueIsGreaterThan 
VAR_INPUT
	(* for the test it's the parameter ``currentValue`` *)
	valueToTest	:LDATE;
	(* for the test it's the parameter ``lessValue`` *)
	lessValue	:LDATE;
END_VAR
VAR
	(* just the expectation if the assertion to test must be worng or true *)
	assertionIsWrong		:BOOL;
	(* contains the format string for the test message *)
	message					:Tc2_System.T_MaxString;
	(* TwinCAT printf with the test message *)
	messageStringBuilder	:Tc2_Utilities.FB_FormatString;
	(* LDATE value of ``currentValue`` as string *)
	currentValueAsString	:STRING(22);
	(* LDATE value of ``lessValue`` as string *)
	lessValueAsString		:STRING(22);
END_VAR
THIS^.assertorContainer.resetAssertor();

assertionIsWrong := (valueToTest <= lessValue);

message := SEL(
	assertionIsWrong,
	'currentValue is %s lessValue is %s assertion must be TRUE', 
	'currentValue is %s lessValue is %s assertion must be FALSE'
);
currentValueAsString := TO_STRING(valueToTest);
lessValueAsString := TO_STRING(lessValue);

messageStringBuilder(
	sFormat := message,
	arg1 := THIS^.AnyToArg(currentValueAsString),
	arg2 := THIS^.AnyToArg(lessValueAsString)
);

THIS^.assertorContainer.assertor.assert.dateAndTime.long.dateOnly.valueIsGreaterThan(
	currentValue	:= valueToTest,
	lessValue		:= lessValue,
	message			:= ''
);

THIS^.AssertEquals_BOOL(
	Expected 	:= assertionIsWrong,
	Actual 		:= THIS^.assertorContainer.wasAssertionWrong,
	Message 	:= messageStringBuilder.sOut
);
END_METHOD

(*

short summary
==================
This test method tests ``assert.dateAndTime.long.dateOnly.valueIsInRangeOf``
method of CNM_AssertionInterfaces library, 
it provides the possibility to handover test data via parameter 


.. <legal notes>

legal notes
=================
| SPDX-FileCopyrightText: © 2022 ekvip automation GmbH <info@ekvip.de>
| SPDX-License-Identifier: Apache-2.0
| For details check: Apache-2.0_

.. _Apache-2.0: https://www.apache.org/licenses/LICENSE-2.0

.. </legal notes>

parameters
==========

*)

METHOD testValueIsInRangeOf 
VAR_INPUT
	(* for the test it's the parameter ``lowerLimit`` *)
	lowerLimit	:LDATE;
	(* for the test it's the parameter ``currentValue`` *)
	valueToTest	:LDATE;
	(* for the test it's the parameter ``upperLimit`` *)
	upperLimit	:LDATE;
END_VAR
VAR
	(* just the expectation if the assertion to test must be worng or true *)
	assertionIsWrong		:BOOL;
	(* contains the format string for the test message *)
	message					:Tc2_System.T_MaxString;
	(* TwinCAT printf with the test message *)
	messageStringBuilder	:Tc2_Utilities.FB_FormatString;
	(* LDATE value of ``lowerLimit`` as string *)
	lowerLimitAsString		:STRING(22);
	(* LDATE value of ``currentValue`` as string *)
	currentValueAsString	:STRING(22);
	(* LDATE value of ``upperLimit`` as string *)
	upperLimitAsString		:STRING(22);

END_VAR
THIS^.assertorContainer.resetAssertor();

assertionIsWrong := ((
		valueToTest < lowerLimit
	) OR (	
		valueToTest > upperLimit
	)
);

message := SEL(
	assertionIsWrong,
	'lowerLimit is %s currentValue is %s upperLimit is %s assertion must be TRUE', 
	'lowerLimit is %s currentValue is %s upperLimit is %s assertion must be FALSE'
);
lowerLimitAsString		:= TO_STRING(lowerLimit);
currentValueAsString	:= TO_STRING(valueToTest);
upperLimitAsString		:= TO_STRING(upperLimit);

messageStringBuilder(
	sFormat := message,
	arg1 := THIS^.AnyToArg(lowerLimitAsString),
	arg2 := THIS^.AnyToArg(currentValueAsString),
	arg3 := THIS^.AnyToArg(upperLimitAsString)
);

THIS^.assertorContainer.assertor.assert.dateAndTime.long.dateOnly.valueIsInRangeOf(
	lowerLimit		:= lowerLimit,
	currentValue	:= valueToTest,
	upperLimit		:= upperLimit,
	message			:= ''
);

THIS^.AssertEquals_BOOL(
	Expected 	:= assertionIsWrong,
	Actual 		:= THIS^.assertorContainer.wasAssertionWrong,
	Message 	:= messageStringBuilder.sOut
);
END_METHOD

(*

short summary
==================
This test method tests ``assert.dateAndTime.long.dateOnly.valueIsLessThan``
method of CNM_AssertionInterfaces library, 
it provides the possibility to handover test data via parameter 


.. <legal notes>

legal notes
=================
| SPDX-FileCopyrightText: © 2022 ekvip automation GmbH <info@ekvip.de>
| SPDX-License-Identifier: Apache-2.0
| For details check: Apache-2.0_

.. _Apache-2.0: https://www.apache.org/licenses/LICENSE-2.0

.. </legal notes>

parameters
==========

*)

METHOD testValueIsLessThan 
VAR_INPUT
	(* for the test it's the parameter ``currentValue`` *)
	valueToTest		:LDATE;
	(* for the test it's the parameter ``greaterValue`` *)
	greaterValue	:LDATE;
END_VAR
VAR
	(* just the expectation if the assertion to test must be worng or true *)
	assertionIsWrong		:BOOL;
	(* contains the format string for the test message *)
	message					:Tc2_System.T_MaxString;
	(* TwinCAT printf with the test message *)
	messageStringBuilder	:Tc2_Utilities.FB_FormatString;
	(* LDATE value of ``currentValue`` as string *)
	currentValueAsString	:STRING(22);
	(* LDATE value of ``greaterValue`` as string *)
	greaterValueAsString	:STRING(22);
END_VAR
THIS^.assertorContainer.resetAssertor();

assertionIsWrong := (valueToTest >= greaterValue);

message := SEL(
	assertionIsWrong,
	'currentValue is %s greaterValue is %s assertion must be TRUE', 
	'currentValue is %s greaterValue is %s assertion must be FALSE'
);
currentValueAsString := TO_STRING(valueToTest);
greaterValueAsString := TO_STRING(greaterValue);

messageStringBuilder(
	sFormat := message,
	arg1 := THIS^.AnyToArg(currentValueAsString),
	arg2 := THIS^.AnyToArg(greaterValueAsString)
);

THIS^.assertorContainer.assertor.assert.dateAndTime.long.dateOnly.valueIsLessThan(
	currentValue	:= valueToTest,
	greaterValue	:= greaterValue,
	message			:= ''
);

THIS^.AssertEquals_BOOL(
	Expected 	:= assertionIsWrong,
	Actual 		:= THIS^.assertorContainer.wasAssertionWrong,
	Message 	:= messageStringBuilder.sOut
);
END_METHOD

(*

short summary
==================
This test method tests ``assert.dateAndTime.long.dateOnly.valueIsMax``
method of CNM_AssertionInterfaces library, 
it provides the possibility to handover test data via parameter 


.. <legal notes>

legal notes
=================
| SPDX-FileCopyrightText: © 2022 ekvip automation GmbH <info@ekvip.de>
| SPDX-License-Identifier: Apache-2.0
| For details check: Apache-2.0_

.. _Apache-2.0: https://www.apache.org/licenses/LICENSE-2.0

.. </legal notes>

parameters
==========

*)

METHOD testValueIsMax 
VAR_INPUT
	(* for the test it's the parameter ``currentValue`` *)
	valueToTest		:LDATE;
	(* for the test it's the parameter ``greaterValue`` *)
	maximumValue	:LDATE;
END_VAR
VAR
	(* just the expectation if the assertion to test must be worng or true *)
	assertionIsWrong		:BOOL;
	(* contains the format string for the test message *)
	message					:Tc2_System.T_MaxString;
	(* TwinCAT printf with the test message *)
	messageStringBuilder	:Tc2_Utilities.FB_FormatString;
	(* LDATE value of ``currentValue`` as string *)
	currentValueAsString	:STRING(22);
	(* LDATE value of ``maximumValue`` as string *)
	maximumValueAsString	:STRING(22);
END_VAR
THIS^.assertorContainer.resetAssertor();

assertionIsWrong := (valueToTest > maximumValue);

message := SEL(
	assertionIsWrong,
	'currentValue is %s maximumValue is %s assertion must be TRUE', 
	'currentValue is %s maximumValue is %s assertion must be FALSE'
);
currentValueAsString := TO_STRING(valueToTest);
maximumValueAsString := TO_STRING(maximumValue);

messageStringBuilder(
	sFormat := message,
	arg1 := THIS^.AnyToArg(currentValueAsString),
	arg2 := THIS^.AnyToArg(maximumValueAsString)
);

THIS^.assertorContainer.assertor.assert.dateAndTime.long.dateOnly.valueIsMax(
	currentValue	:= valueToTest,
	maximumValue	:= maximumValue,
	message			:= ''
);

THIS^.AssertEquals_BOOL(
	Expected 	:= assertionIsWrong,
	Actual 		:= THIS^.assertorContainer.wasAssertionWrong,
	Message 	:= messageStringBuilder.sOut
);
END_METHOD

(*

short summary
==================
This test method tests ``assert.dateAndTime.long.dateOnly.valueIsMin``
method of CNM_AssertionInterfaces library, 
it provides the possibility to handover test data via parameter 


.. <legal notes>

legal notes
=================
| SPDX-FileCopyrightText: © 2022 ekvip automation GmbH <info@ekvip.de>
| SPDX-License-Identifier: Apache-2.0
| For details check: Apache-2.0_

.. _Apache-2.0: https://www.apache.org/licenses/LICENSE-2.0

.. </legal notes>

parameters
==========

*)

METHOD testValueIsMin 
VAR_INPUT
	(* for the test it's the parameter ``currentValue`` *)
	valueToTest		:LDATE;
	(* for the test it's the parameter ``greaterValue`` *)
	minimumValue	:LDATE;
END_VAR
VAR
	(* just the expectation if the assertion to test must be worng or true *)
	assertionIsWrong		:BOOL;
	(* contains the format string for the test message *)
	message					:Tc2_System.T_MaxString;
	(* TwinCAT printf with the test message *)
	messageStringBuilder	:Tc2_Utilities.FB_FormatString;
	(* LDATE value of ``currentValue`` as string *)
	currentValueAsString	:STRING(22);
	(* LDATE value of ``minimumValue`` as string *)
	minimumValueAsString	:STRING(22);
END_VAR
THIS^.assertorContainer.resetAssertor();

assertionIsWrong := (valueToTest < minimumValue);

message := SEL(
	assertionIsWrong,
	'currentValue is %s minimumValue is %s assertion must be TRUE', 
	'currentValue is %s minimumValue is %s assertion must be FALSE'
);
currentValueAsString := TO_STRING(valueToTest);
minimumValueAsString := TO_STRING(minimumValue);

messageStringBuilder(
	sFormat := message,
	arg1 := THIS^.AnyToArg(currentValueAsString),
	arg2 := THIS^.AnyToArg(minimumValueAsString)
);

THIS^.assertorContainer.assertor.assert.dateAndTime.long.dateOnly.valueIsMin(
	currentValue	:= valueToTest,
	minimumValue	:= minimumValue,
	message			:= ''
);

THIS^.AssertEquals_BOOL(
	Expected 	:= assertionIsWrong,
	Actual 		:= THIS^.assertorContainer.wasAssertionWrong,
	Message 	:= messageStringBuilder.sOut
);
END_METHOD

(*

short summary
==================
This test method tests ``assert.dateAndTime.long.dateOnly.valueIsNotEqualTo``
method of CNM_AssertionInterfaces library, 
it provides the possibility to handover test data via parameter 


.. <legal notes>

legal notes
=================
| SPDX-FileCopyrightText: © 2022 ekvip automation GmbH <info@ekvip.de>
| SPDX-License-Identifier: Apache-2.0
| For details check: Apache-2.0_

.. _Apache-2.0: https://www.apache.org/licenses/LICENSE-2.0

.. </legal notes>

parameters
==========

*)

METHOD testValueIsNotEqualTo 
VAR_INPUT
	(* for the test it's the parameter ``currentValue`` *)
	valueToTest		:LDATE;
	(* for the test it's the parameter ``unexpectedValue`` *)
	unexpectedValue	:LDATE;
END_VAR
VAR
	(* just the expectation if the assertion to test must be worng or true *)
	assertionIsWrong		:BOOL;
	(* contains the format string for the test message *)
	message					:Tc2_System.T_MaxString;
	(* TwinCAT printf with the test message *)
	messageStringBuilder	:Tc2_Utilities.FB_FormatString;
	(* LDATE value of ``currentValue`` as string *)
	currentValueAsString	:STRING(22);
	(* LDATE value of ``unexpectedValue`` as string *)
	unexpectedValueAsString	:STRING(22);
END_VAR
THIS^.assertorContainer.resetAssertor();

assertionIsWrong := (valueToTest = unexpectedValue);
message := SEL(
	assertionIsWrong,
	'currentValue is %s expectedValue is %s assertion must be TRUE', 
	'currentValue is %s expectedValue is %s assertion must be FALSE'
);
currentValueAsString := TO_STRING(valueToTest);
unexpectedValueAsString := TO_STRING(unexpectedValue);

messageStringBuilder(
	sFormat := message,
	arg1 := THIS^.AnyToArg(currentValueAsString),
	arg2 := THIS^.AnyToArg(unexpectedValueAsString)
);

THIS^.assertorContainer.assertor.assert.dateAndTime.long.dateOnly.valueIsNotEqualTo(
	currentValue	:= valueToTest,
	unexpectedValue	:= unexpectedValue,
	message			:= ''
);

THIS^.AssertEquals_BOOL(
	Expected 	:= assertionIsWrong,
	Actual 		:= THIS^.assertorContainer.wasAssertionWrong,
	Message 	:= messageStringBuilder.sOut
);
END_METHOD

END_FUNCTION_BLOCK

// ---- AssertionTester/AssertionTests/DateTimeAssertions/classes/LDTAssertionTests.TcPOU
(*

short summary
==================
This class tests all methods of LDT assertions
with various combinations of inputs and checks expected 
outputs are satisfied or not

.. <legal notes>

legal notes
=================
| SPDX-FileCopyrightText: © 2022 ekvip automation GmbH <info@ekvip.de>
| SPDX-License-Identifier: Apache-2.0
| For details check: Apache-2.0_

.. _Apache-2.0: https://www.apache.org/licenses/LICENSE-2.0

.. </legal notes>

methods and properties
======================

*)


FUNCTION_BLOCK LDTAssertionTests EXTENDS AbstractAssertorTest
VAR
	
END_VAR
VAR CONSTANT
	(* prefix to unify the test names *)
	TEST_NAME_PREFIX		:STRING := 'assert.dateAndTime.long.dateAndTime.';
	(* max value of a LWORD *)
	{attribute 'hide'}
	MAX_LWORD				:LWORD := 16#FFFF_FFFF_FFFF_FFFF;
	(* min value of a LWORD *)
	{attribute 'hide'}
	MIN_LWORD				:LWORD := 16#0000_0000_0000_0000;
	(* only the msb is set *)
	{attribute 'hide'}
	MSB_ONLY				:LWORD := 16#8000_0000_0000_0000;
	(* only the msb is set *)
	{attribute 'hide'}
	LSB_ONLY				:LWORD := 16#0000_0000_0000_0001;
	(* all bits set except the msb *)
	{attribute 'hide'}
	WITHOUT_MSB 			:LWORD := 16#7FFF_FFFF_FFFF_FFFF;
	(* for every nibble is the msb set only *)
	{attribute 'hide'}
	ALL_NIBBLE_MSB			:LWORD := 16#8888_8888_8888_8888;
	(* for every nibble is the msb unset only *)
	{attribute 'hide'}
	WITHOUT_NIBBLE_MSB		:LWORD := 16#7777_7777_7777_7777;
	(* for every nibble is the lsb set only *)
	{attribute 'hide'}
	ALL_NIBBLE_LSB			:LWORD := 16#1111_1111_1111_1111;
	(* every bit is set except the lsb *)
	{attribute 'hide'}
	LSB_IS_UNSET			:LWORD := 16#FFFF__FFFF_FFFF_FFFE;
	(* max vale of date and time *)
	LDT_MAX					:LDT := TO_LDT(MAX_LWORD);
	(* min vale of date and time *)
	LDT_MIN					:LDT := TO_LDT(MIN_LWORD);
	(* only the msb is set *)
	LDT_MSB_ONLY			:LDT := TO_LDT(MSB_ONLY);
	(* all bits set except the msb *)
	LDT_WITHOUT_MSB 		:LDT := TO_LDT(WITHOUT_MSB);
	(* for every nibble is the msb set only *)
	LDT_ALL_NIBBLE_MSB		:LDT := TO_LDT(ALL_NIBBLE_MSB);
	(* for every nibble is the msb unset only *)
	LDT_WITHOUT_NIBBLE_MSB	:LDT := TO_LDT(WITHOUT_NIBBLE_MSB);
	(* for every nibble is the lsb set only *)
	LDT_ALL_NIBBLE_LSB		:LDT := TO_LDT(ALL_NIBBLE_LSB);	
	(* every bit is set except the lsb *)
	LDT_LSB_IS_UNSET		:LDT := TO_LDT(LSB_IS_UNSET);
	(* only the msb is set *)
	LDT_LSB_ONLY			:LDT := TO_LDT(LSB_ONLY);
END_VAR

THIS^.runValueIsEqualToTests();
THIS^.runValueIsGreaterThanTests();
THIS^.runValueIsInRangeOfTests();
THIS^.runValueIsLessThanTests();
THIS^.runValueIsMaxTests();
THIS^.runValueIsMinTests();
THIS^.runValueIsNotEqualToTests();

(*

short summary
==================
This test method is a helper function to create a unified test name

.. <legal notes>

legal notes
=================
| SPDX-FileCopyrightText: © 2022 ekvip automation GmbH <info@ekvip.de>
| SPDX-License-Identifier: Apache-2.0
| For details check: Apache-2.0_

.. _Apache-2.0: https://www.apache.org/licenses/LICENSE-2.0

.. </legal notes>

parameters
==========

*)

METHOD PROTECTED getTestNameFor :Tc2_System.T_MaxString
VAR_INPUT
	(* name of the method to test, to create a unified test name *)
	nameOfMethodToTest	:Tc2_System.T_MaxString;
END_VAR
getTestNameFor := Tc2_Standard.CONCAT(THIS^.TEST_NAME_PREFIX, nameOfMethodToTest);
END_METHOD

(*

short summary
==================
This test method tests ``assert.dateAndTime.long.dateAndTime.valueIsEqualTo``
method of CNM_AssertionInterfaces library with various inputs

.. <legal notes>

legal notes
=================
| SPDX-FileCopyrightText: © 2022 ekvip automation GmbH <info@ekvip.de>
| SPDX-License-Identifier: Apache-2.0
| For details check: Apache-2.0_

.. _Apache-2.0: https://www.apache.org/licenses/LICENSE-2.0

.. </legal notes>

*)

METHOD runValueIsEqualToTests
RETURN (NOT TcUnit.TEST_ORDERED(THIS^.getTestNameFor('valueIsEqualTo')));

THIS^.testValueIsEqualTo(
	valueToTest := THIS^.LDT_MAX,
	expected := THIS^.LDT_MAX
);
THIS^.testValueIsEqualTo(
	valueToTest := THIS^.LDT_MIN,
	expected := THIS^.LDT_MIN
);
THIS^.testValueIsEqualTo(
	valueToTest := THIS^.LDT_MIN,
	expected := THIS^.LDT_MAX
);
THIS^.testValueIsEqualTo(
	valueToTest := THIS^.LDT_MAX,
	expected := THIS^.LDT_MIN
);
THIS^.testValueIsEqualTo(
	valueToTest := THIS^.LDT_ALL_NIBBLE_LSB,
	expected := THIS^.LDT_ALL_NIBBLE_LSB
);
THIS^.testValueIsEqualTo(
	valueToTest := THIS^.LDT_LSB_ONLY,
	expected := THIS^.LDT_MSB_ONLY
);
THIS^.testValueIsEqualTo(
	valueToTest := THIS^.LDT_MSB_ONLY,
	expected := THIS^.LDT_MSB_ONLY
);
THIS^.testValueIsEqualTo(
	valueToTest := THIS^.LDT_MSB_ONLY,
	expected := THIS^.LDT_LSB_ONLY
);

TcUnit.TEST_FINISHED();
END_METHOD

(*

short summary
==================
This test method tests ``assert.dateAndTime.long.dateAndTime.valueIsGreaterThan``
method of CNM_AssertionInterfaces library with various inputs

.. <legal notes>

legal notes
=================
| SPDX-FileCopyrightText: © 2022 ekvip automation GmbH <info@ekvip.de>
| SPDX-License-Identifier: Apache-2.0
| For details check: Apache-2.0_

.. _Apache-2.0: https://www.apache.org/licenses/LICENSE-2.0

.. </legal notes>

*)

METHOD runValueIsGreaterThanTests
RETURN (NOT TcUnit.TEST_ORDERED(THIS^.getTestNameFor('valueIsGreaterThan')));

THIS^.testValueIsGreaterThan(
	valueToTest := THIS^.LDT_MAX,
	lessValue := THIS^.LDT_MAX
);
THIS^.testValueIsGreaterThan(
	valueToTest := THIS^.LDT_MIN,
	lessValue := THIS^.LDT_MIN
);
THIS^.testValueIsGreaterThan(
	valueToTest := THIS^.LDT_MIN,
	lessValue := THIS^.LDT_MAX
);
THIS^.testValueIsGreaterThan(
	valueToTest := THIS^.LDT_MAX,
	lessValue := THIS^.LDT_MIN
);
THIS^.testValueIsGreaterThan(
	valueToTest := THIS^.LDT_ALL_NIBBLE_LSB,
	lessValue := THIS^.LDT_ALL_NIBBLE_LSB
);
THIS^.testValueIsGreaterThan(
	valueToTest := THIS^.LDT_ALL_NIBBLE_MSB,
	lessValue := THIS^.LDT_ALL_NIBBLE_LSB
);
THIS^.testValueIsGreaterThan(
	valueToTest := THIS^.LDT_ALL_NIBBLE_LSB,
	lessValue := THIS^.LDT_ALL_NIBBLE_MSB
);
THIS^.testValueIsGreaterThan(
	valueToTest := THIS^.LDT_LSB_ONLY,
	lessValue := THIS^.LDT_MSB_ONLY
);
THIS^.testValueIsGreaterThan(
	valueToTest := THIS^.LDT_MSB_ONLY,
	lessValue := THIS^.LDT_MSB_ONLY
);
THIS^.testValueIsGreaterThan(
	valueToTest := THIS^.LDT_MSB_ONLY,
	lessValue := THIS^.LDT_LSB_ONLY
);
THIS^.testValueIsGreaterThan(
	valueToTest := THIS^.LDT_LSB_IS_UNSET,
	lessValue := THIS^.LDT_MAX
);
THIS^.testValueIsGreaterThan(
	valueToTest := THIS^.LDT_MAX,
	lessValue := THIS^.LDT_LSB_IS_UNSET
);

TcUnit.TEST_FINISHED();
END_METHOD

(*

short summary
==================
This test method tests ``assert.dateAndTime.long.dateAndTime.valueIsInRangeOf``
method of CNM_AssertionInterfaces library with various inputs

.. <legal notes>

legal notes
=================
| SPDX-FileCopyrightText: © 2022 ekvip automation GmbH <info@ekvip.de>
| SPDX-License-Identifier: Apache-2.0
| For details check: Apache-2.0_

.. _Apache-2.0: https://www.apache.org/licenses/LICENSE-2.0

.. </legal notes>

*)

METHOD runValueIsInRangeOfTests
RETURN (NOT TcUnit.TEST_ORDERED(THIS^.getTestNameFor('valueIsInRangeOf')));

THIS^.testValueIsInRangeOf(
	lowerLimit := THIS^.LDT_MIN,
	valueToTest := THIS^.LDT_MAX,
	upperLimit	:= THIS^.LDT_MAX
);
THIS^.testValueIsInRangeOf(
	lowerLimit := THIS^.LDT_MIN,
	valueToTest := THIS^.LDT_MIN,
	upperLimit	:= THIS^.LDT_MAX
);
THIS^.testValueIsInRangeOf(
	lowerLimit := THIS^.LDT_MAX,
	valueToTest := THIS^.LDT_MAX,
	upperLimit	:= THIS^.LDT_MIN
);
THIS^.testValueIsInRangeOf(
	lowerLimit := THIS^.LDT_MAX,
	valueToTest := THIS^.LDT_MIN,
	upperLimit	:= THIS^.LDT_MIN
);
THIS^.testValueIsInRangeOf(
	lowerLimit := THIS^.LDT_LSB_IS_UNSET,
	valueToTest := THIS^.LDT_MIN,
	upperLimit	:= THIS^.LDT_MAX
);
THIS^.testValueIsInRangeOf(
	lowerLimit := THIS^.LDT_MIN,
	valueToTest := THIS^.LDT_LSB_IS_UNSET,
	upperLimit	:= THIS^.LDT_MAX
);
THIS^.testValueIsInRangeOf(
	lowerLimit := THIS^.LDT_LSB_IS_UNSET,
	valueToTest := THIS^.LDT_LSB_IS_UNSET,
	upperLimit	:= THIS^.LDT_LSB_IS_UNSET
);
THIS^.testValueIsInRangeOf(
	lowerLimit := THIS^.LDT_ALL_NIBBLE_LSB,
	valueToTest := THIS^.LDT_LSB_IS_UNSET,
	upperLimit	:= THIS^.LDT_ALL_NIBBLE_MSB
);
THIS^.testValueIsInRangeOf(
	lowerLimit := THIS^.LDT_LSB_IS_UNSET,
	valueToTest := THIS^.LDT_ALL_NIBBLE_LSB,
	upperLimit	:= THIS^.LDT_ALL_NIBBLE_MSB
);
THIS^.testValueIsInRangeOf(
	lowerLimit := THIS^.LDT_LSB_ONLY,
	valueToTest := THIS^.LDT_WITHOUT_MSB,
	upperLimit	:= THIS^.LDT_MSB_ONLY
);
THIS^.testValueIsInRangeOf(
	lowerLimit := THIS^.LDT_WITHOUT_MSB,
	valueToTest := THIS^.LDT_LSB_ONLY,
	upperLimit	:= THIS^.LDT_MSB_ONLY
);
THIS^.testValueIsInRangeOf(
	lowerLimit := THIS^.LDT_WITHOUT_NIBBLE_MSB,
	valueToTest := THIS^.LDT_MAX,
	upperLimit	:= THIS^.LDT_ALL_NIBBLE_MSB
);
THIS^.testValueIsInRangeOf(
	lowerLimit := THIS^.LDT_WITHOUT_NIBBLE_MSB,
	valueToTest := THIS^.LDT_MIN,
	upperLimit	:= THIS^.LDT_ALL_NIBBLE_MSB
);
THIS^.testValueIsInRangeOf(
	lowerLimit := THIS^.LDT_WITHOUT_NIBBLE_MSB,
	valueToTest := THIS^.LDT_WITHOUT_NIBBLE_MSB,
	upperLimit	:= THIS^.LDT_ALL_NIBBLE_MSB
);
THIS^.testValueIsInRangeOf(
	lowerLimit := THIS^.LDT_WITHOUT_NIBBLE_MSB,
	valueToTest := THIS^.LDT_ALL_NIBBLE_MSB,
	upperLimit	:= THIS^.LDT_ALL_NIBBLE_MSB
);

TcUnit.TEST_FINISHED();
END_METHOD

(*

short summary
==================
This test method tests ``assert.dateAndTime.long.dateAndTime.valueIsLessThan``
method of CNM_AssertionInterfaces library with various inputs

.. <legal notes>

legal notes
=================
| SPDX-FileCopyrightText: © 2022 ekvip automation GmbH <info@ekvip.de>
| SPDX-License-Identifier: Apache-2.0
| For details check: Apache-2.0_

.. _Apache-2.0: https://www.apache.org/licenses/LICENSE-2.0

.. </legal notes>

*)

METHOD runValueIsLessThanTests
RETURN (NOT TcUnit.TEST_ORDERED(THIS^.getTestNameFor('valueIsLessThan')));

THIS^.testValueIsLessThan(
	valueToTest := THIS^.LDT_MAX,
	greaterValue := THIS^.LDT_MAX
);
THIS^.testValueIsLessThan(
	valueToTest := THIS^.LDT_MIN,
	greaterValue := THIS^.LDT_MIN
);
THIS^.testValueIsLessThan(
	valueToTest := THIS^.LDT_MIN,
	greaterValue := THIS^.LDT_MAX
);
THIS^.testValueIsLessThan(
	valueToTest := THIS^.LDT_MAX,
	greaterValue := THIS^.LDT_MIN
);
THIS^.testValueIsLessThan(
	valueToTest := THIS^.LDT_ALL_NIBBLE_LSB,
	greaterValue := THIS^.LDT_ALL_NIBBLE_LSB
);
THIS^.testValueIsLessThan(
	valueToTest := THIS^.LDT_ALL_NIBBLE_MSB,
	greaterValue := THIS^.LDT_ALL_NIBBLE_LSB
);
THIS^.testValueIsLessThan(
	valueToTest := THIS^.LDT_ALL_NIBBLE_LSB,
	greaterValue := THIS^.LDT_ALL_NIBBLE_MSB
);
THIS^.testValueIsLessThan(
	valueToTest := THIS^.LDT_LSB_ONLY,
	greaterValue := THIS^.LDT_MSB_ONLY
);
THIS^.testValueIsLessThan(
	valueToTest := THIS^.LDT_MSB_ONLY,
	greaterValue := THIS^.LDT_MSB_ONLY
);
THIS^.testValueIsLessThan(
	valueToTest := THIS^.LDT_MSB_ONLY,
	greaterValue := THIS^.LDT_LSB_ONLY
);
THIS^.testValueIsLessThan(
	valueToTest := THIS^.LDT_LSB_IS_UNSET,
	greaterValue := THIS^.LDT_MAX
);
THIS^.testValueIsLessThan(
	valueToTest := THIS^.LDT_MAX,
	greaterValue := THIS^.LDT_LSB_IS_UNSET
);

TcUnit.TEST_FINISHED();
END_METHOD

(*

short summary
==================
This test method tests ``assert.dateAndTime.long.dateAndTime.valueIsMax``
method of CNM_AssertionInterfaces library with various inputs

.. <legal notes>

legal notes
=================
| SPDX-FileCopyrightText: © 2022 ekvip automation GmbH <info@ekvip.de>
| SPDX-License-Identifier: Apache-2.0
| For details check: Apache-2.0_

.. _Apache-2.0: https://www.apache.org/licenses/LICENSE-2.0

.. </legal notes>

*)

METHOD runValueIsMaxTests
RETURN (NOT TcUnit.TEST_ORDERED(THIS^.getTestNameFor('valueIsMax')));

THIS^.testValueIsMax(
	valueToTest := THIS^.LDT_MAX,
	maximumValue := THIS^.LDT_MAX
);
THIS^.testValueIsMax(
	valueToTest := THIS^.LDT_MIN,
	maximumValue := THIS^.LDT_MIN
);
THIS^.testValueIsMax(
	valueToTest := THIS^.LDT_MIN,
	maximumValue := THIS^.LDT_MAX
);
THIS^.testValueIsMax(
	valueToTest := THIS^.LDT_MAX,
	maximumValue := THIS^.LDT_MIN
);
THIS^.testValueIsMax(
	valueToTest := THIS^.LDT_ALL_NIBBLE_LSB,
	maximumValue := THIS^.LDT_ALL_NIBBLE_LSB
);
THIS^.testValueIsMax(
	valueToTest := THIS^.LDT_ALL_NIBBLE_MSB,
	maximumValue := THIS^.LDT_ALL_NIBBLE_LSB
);
THIS^.testValueIsMax(
	valueToTest := THIS^.LDT_ALL_NIBBLE_LSB,
	maximumValue := THIS^.LDT_ALL_NIBBLE_MSB
);
THIS^.testValueIsMax(
	valueToTest := THIS^.LDT_LSB_ONLY,
	maximumValue := THIS^.LDT_MSB_ONLY
);
THIS^.testValueIsMax(
	valueToTest := THIS^.LDT_MSB_ONLY,
	maximumValue := THIS^.LDT_MSB_ONLY
);
THIS^.testValueIsMax(
	valueToTest := THIS^.LDT_MSB_ONLY,
	maximumValue := THIS^.LDT_LSB_ONLY
);
THIS^.testValueIsMax(
	valueToTest := THIS^.LDT_LSB_IS_UNSET,
	maximumValue := THIS^.LDT_MAX
);
THIS^.testValueIsMax(
	valueToTest := THIS^.LDT_MAX,
	maximumValue := THIS^.LDT_LSB_IS_UNSET
);

TcUnit.TEST_FINISHED();
END_METHOD

(*

short summary
==================
This test method tests ``assert.dateAndTime.long.dateAndTime.valueIsMin``
method of CNM_AssertionInterfaces library with various inputs

.. <legal notes>

legal notes
=================
| SPDX-FileCopyrightText: © 2022 ekvip automation GmbH <info@ekvip.de>
| SPDX-License-Identifier: Apache-2.0
| For details check: Apache-2.0_

.. _Apache-2.0: https://www.apache.org/licenses/LICENSE-2.0

.. </legal notes>

*)

METHOD runValueIsMinTests
RETURN (NOT TcUnit.TEST_ORDERED(THIS^.getTestNameFor('valueIsMin')));

THIS^.testValueIsMin(
	valueToTest := THIS^.LDT_MAX,
	minimumValue := THIS^.LDT_MAX
);
THIS^.testValueIsMin(
	valueToTest := THIS^.LDT_MIN,
	minimumValue := THIS^.LDT_MIN
);
THIS^.testValueIsMin(
	valueToTest := THIS^.LDT_MIN,
	minimumValue := THIS^.LDT_MAX
);
THIS^.testValueIsMin(
	valueToTest := THIS^.LDT_MAX,
	minimumValue := THIS^.LDT_MIN
);
THIS^.testValueIsMin(
	valueToTest := THIS^.LDT_ALL_NIBBLE_LSB,
	minimumValue := THIS^.LDT_ALL_NIBBLE_LSB
);
THIS^.testValueIsMin(
	valueToTest := THIS^.LDT_ALL_NIBBLE_MSB,
	minimumValue := THIS^.LDT_ALL_NIBBLE_LSB
);
THIS^.testValueIsMin(
	valueToTest := THIS^.LDT_ALL_NIBBLE_LSB,
	minimumValue := THIS^.LDT_ALL_NIBBLE_MSB
);
THIS^.testValueIsMin(
	valueToTest := THIS^.LDT_LSB_ONLY,
	minimumValue := THIS^.LDT_MSB_ONLY
);
THIS^.testValueIsMin(
	valueToTest := THIS^.LDT_MSB_ONLY,
	minimumValue := THIS^.LDT_MSB_ONLY
);
THIS^.testValueIsMin(
	valueToTest := THIS^.LDT_MSB_ONLY,
	minimumValue := THIS^.LDT_LSB_ONLY
);
THIS^.testValueIsMin(
	valueToTest := THIS^.LDT_LSB_IS_UNSET,
	minimumValue := THIS^.LDT_MAX
);
THIS^.testValueIsMin(
	valueToTest := THIS^.LDT_MAX,
	minimumValue := THIS^.LDT_LSB_IS_UNSET
);

TcUnit.TEST_FINISHED();
END_METHOD

(*

short summary
==================
This test method tests ``assert.dateAndTime.long.dateAndTime.valueIsNotEqualTo``
method of CNM_AssertionInterfaces library with various inputs

.. <legal notes>

legal notes
=================
| SPDX-FileCopyrightText: © 2022 ekvip automation GmbH <info@ekvip.de>
| SPDX-License-Identifier: Apache-2.0
| For details check: Apache-2.0_

.. _Apache-2.0: https://www.apache.org/licenses/LICENSE-2.0

.. </legal notes>

*)

METHOD runValueIsNotEqualToTests
RETURN (NOT TcUnit.TEST_ORDERED(THIS^.getTestNameFor('valueIsNotEqualTo')));

THIS^.testValueIsNotEqualTo(
	valueToTest := THIS^.LDT_MAX,
	unexpectedValue := THIS^.LDT_MAX
);
THIS^.testValueIsNotEqualTo(
	valueToTest := THIS^.LDT_MIN,
	unexpectedValue := THIS^.LDT_MIN
);
THIS^.testValueIsNotEqualTo(
	valueToTest := THIS^.LDT_MIN,
	unexpectedValue := THIS^.LDT_MAX
);
THIS^.testValueIsNotEqualTo(
	valueToTest := THIS^.LDT_MAX,
	unexpectedValue := THIS^.LDT_MIN
);
THIS^.testValueIsNotEqualTo(
	valueToTest := THIS^.LDT_ALL_NIBBLE_LSB,
	unexpectedValue := THIS^.LDT_ALL_NIBBLE_LSB
);
THIS^.testValueIsNotEqualTo(
	valueToTest := THIS^.LDT_LSB_ONLY,
	unexpectedValue := THIS^.LDT_MSB_ONLY
);
THIS^.testValueIsNotEqualTo(
	valueToTest := THIS^.LDT_MSB_ONLY,
	unexpectedValue := THIS^.LDT_MSB_ONLY
);
THIS^.testValueIsNotEqualTo(
	valueToTest := THIS^.LDT_MSB_ONLY,
	unexpectedValue := THIS^.LDT_LSB_ONLY
);

TcUnit.TEST_FINISHED();
END_METHOD

(*

short summary
==================
This test method tests ``assert.dateAndTime.long.dateAndTime.valueIsEqualTo``
method of CNM_AssertionInterfaces library, 
it provides the possibility to handover test data via parameter 


.. <legal notes>

legal notes
=================
| SPDX-FileCopyrightText: © 2022 ekvip automation GmbH <info@ekvip.de>
| SPDX-License-Identifier: Apache-2.0
| For details check: Apache-2.0_

.. _Apache-2.0: https://www.apache.org/licenses/LICENSE-2.0

.. </legal notes>

parameters
==========

*)

METHOD testValueIsEqualTo 
VAR_INPUT
	(* for the test it's the parameter ``currentValue`` *)
	valueToTest	:LDT;
	(* for the test it's the parameter ``expectedValue`` *)
	expected	:LDT;
END_VAR
VAR
	(* just the expectation if the assertion to test must be worng or true *)
	assertionIsWrong		:BOOL;
	(* contains the format string for the test message *)
	message					:Tc2_System.T_MaxString;
	(* TwinCAT printf with the test message *)
	messageStringBuilder	:Tc2_Utilities.FB_FormatString;
	(* LDT value of ``currentValue`` as string *)
	currentValueAsString	:STRING(22);
	(* LDT value of ``expectedValue`` as string *)
	expectedValueAsString	:STRING(22);
END_VAR
THIS^.assertorContainer.resetAssertor();

assertionIsWrong := (valueToTest <> expected);

message := SEL(
	assertionIsWrong,
	'currentValue is %s expectedValue is %s assertion must be TRUE', 
	'currentValue is %s expectedValue is %s assertion must be FALSE'
);
currentValueAsString := TO_STRING(valueToTest);
expectedValueAsString := TO_STRING(expected);

messageStringBuilder(
	sFormat := message,
	arg1 := THIS^.AnyToArg(currentValueAsString),
	arg2 := THIS^.AnyToArg(expectedValueAsString)
);

THIS^.assertorContainer.assertor.assert.dateAndTime.long.dateAndTime.valueIsEqualTo(
	currentValue	:= valueToTest,
	expectedValue	:= expected,
	message			:= ''
);

THIS^.AssertEquals_BOOL(
	Expected 	:= assertionIsWrong,
	Actual 		:= THIS^.assertorContainer.wasAssertionWrong,
	Message 	:= messageStringBuilder.sOut
);
END_METHOD

(*

short summary
==================
This test method tests ``assert.dateAndTime.long.dateAndTime.valueIsGreaterThan``
method of CNM_AssertionInterfaces library, 
it provides the possibility to handover test data via parameter 


.. <legal notes>

legal notes
=================
| SPDX-FileCopyrightText: © 2022 ekvip automation GmbH <info@ekvip.de>
| SPDX-License-Identifier: Apache-2.0
| For details check: Apache-2.0_

.. _Apache-2.0: https://www.apache.org/licenses/LICENSE-2.0

.. </legal notes>

parameters
==========

*)

METHOD testValueIsGreaterThan 
VAR_INPUT
	(* for the test it's the parameter ``currentValue`` *)
	valueToTest	:LDT;
	(* for the test it's the parameter ``lessValue`` *)
	lessValue	:LDT;
END_VAR
VAR
	(* just the expectation if the assertion to test must be worng or true *)
	assertionIsWrong		:BOOL;
	(* contains the format string for the test message *)
	message					:Tc2_System.T_MaxString;
	(* TwinCAT printf with the test message *)
	messageStringBuilder	:Tc2_Utilities.FB_FormatString;
	(* LDT value of ``currentValue`` as string *)
	currentValueAsString	:STRING(22);
	(* LDT value of ``lessValue`` as string *)
	lessValueAsString		:STRING(22);
END_VAR
THIS^.assertorContainer.resetAssertor();

assertionIsWrong := (valueToTest <= lessValue);

message := SEL(
	assertionIsWrong,
	'currentValue is %s lessValue is %s assertion must be TRUE', 
	'currentValue is %s lessValue is %s assertion must be FALSE'
);
currentValueAsString := TO_STRING(valueToTest);
lessValueAsString := TO_STRING(lessValue);

messageStringBuilder(
	sFormat := message,
	arg1 := THIS^.AnyToArg(currentValueAsString),
	arg2 := THIS^.AnyToArg(lessValueAsString)
);

THIS^.assertorContainer.assertor.assert.dateAndTime.long.dateAndTime.valueIsGreaterThan(
	currentValue	:= valueToTest,
	lessValue		:= lessValue,
	message			:= ''
);

THIS^.AssertEquals_BOOL(
	Expected 	:= assertionIsWrong,
	Actual 		:= THIS^.assertorContainer.wasAssertionWrong,
	Message 	:= messageStringBuilder.sOut
);
END_METHOD

(*

short summary
==================
This test method tests ``assert.dateAndTime.long.dateAndTime.valueIsInRangeOf``
method of CNM_AssertionInterfaces library, 
it provides the possibility to handover test data via parameter 


.. <legal notes>

legal notes
=================
| SPDX-FileCopyrightText: © 2022 ekvip automation GmbH <info@ekvip.de>
| SPDX-License-Identifier: Apache-2.0
| For details check: Apache-2.0_

.. _Apache-2.0: https://www.apache.org/licenses/LICENSE-2.0

.. </legal notes>

parameters
==========

*)

METHOD testValueIsInRangeOf 
VAR_INPUT
	(* for the test it's the parameter ``lowerLimit`` *)
	lowerLimit	:LDT;
	(* for the test it's the parameter ``currentValue`` *)
	valueToTest	:LDT;
	(* for the test it's the parameter ``upperLimit`` *)
	upperLimit	:LDT;
END_VAR
VAR
	(* just the expectation if the assertion to test must be worng or true *)
	assertionIsWrong		:BOOL;
	(* contains the format string for the test message *)
	message					:Tc2_System.T_MaxString;
	(* TwinCAT printf with the test message *)
	messageStringBuilder	:Tc2_Utilities.FB_FormatString;
	(* LDT value of ``lowerLimit`` as string *)
	lowerLimitAsString		:STRING(22);
	(* LDT value of ``currentValue`` as string *)
	currentValueAsString	:STRING(22);
	(* dt value of ``upperLimit`` as string *)
	upperLimitAsString		:STRING(22);

END_VAR
THIS^.assertorContainer.resetAssertor();

assertionIsWrong := ((
		valueToTest < lowerLimit
	) OR (
		valueToTest > upperLimit
	)
);

message := SEL(
	assertionIsWrong,
	'lowerLimit is %s currentValue is %s upperLimit is %s assertion must be TRUE', 
	'lowerLimit is %s currentValue is %s upperLimit is %s assertion must be FALSE'
);
lowerLimitAsString		:= TO_STRING(lowerLimit);
currentValueAsString	:= TO_STRING(valueToTest);
upperLimitAsString		:= TO_STRING(upperLimit);

messageStringBuilder(
	sFormat := message,
	arg1 := THIS^.AnyToArg(lowerLimitAsString),
	arg2 := THIS^.AnyToArg(currentValueAsString),
	arg3 := THIS^.AnyToArg(upperLimitAsString)
);

THIS^.assertorContainer.assertor.assert.dateAndTime.long.dateAndTime.valueIsInRangeOf(
	lowerLimit		:= lowerLimit,
	currentValue	:= valueToTest,
	upperLimit		:= upperLimit,
	message			:= ''
);

THIS^.AssertEquals_BOOL(
	Expected 	:= assertionIsWrong,
	Actual 		:= THIS^.assertorContainer.wasAssertionWrong,
	Message 	:= messageStringBuilder.sOut
);
END_METHOD

(*

short summary
==================
This test method tests ``assert.dateAndTime.long.dateAndTime.valueIsLessThan``
method of CNM_AssertionInterfaces library, 
it provides the possibility to handover test data via parameter 


.. <legal notes>

legal notes
=================
| SPDX-FileCopyrightText: © 2022 ekvip automation GmbH <info@ekvip.de>
| SPDX-License-Identifier: Apache-2.0
| For details check: Apache-2.0_

.. _Apache-2.0: https://www.apache.org/licenses/LICENSE-2.0

.. </legal notes>

parameters
==========

*)

METHOD testValueIsLessThan 
VAR_INPUT
	(* for the test it's the parameter ``currentValue`` *)
	valueToTest		:LDT;
	(* for the test it's the parameter ``greaterValue`` *)
	greaterValue	:LDT;
END_VAR
VAR
	(* just the expectation if the assertion to test must be worng or true *)
	assertionIsWrong		:BOOL;
	(* contains the format string for the test message *)
	message					:Tc2_System.T_MaxString;
	(* TwinCAT printf with the test message *)
	messageStringBuilder	:Tc2_Utilities.FB_FormatString;
	(* LDT value of ``currentValue`` as string *)
	currentValueAsString	:STRING(22);
	(* LDT value of ``greaterValue`` as string *)
	greaterValueAsString	:STRING(22);
END_VAR
THIS^.assertorContainer.resetAssertor();

assertionIsWrong := (valueToTest >= greaterValue);

message := SEL(
	assertionIsWrong,
	'currentValue is %s greaterValue is %s assertion must be TRUE', 
	'currentValue is %s greaterValue is %s assertion must be FALSE'
);
currentValueAsString := TO_STRING(valueToTest);
greaterValueAsString := TO_STRING(greaterValue);

messageStringBuilder(
	sFormat := message,
	arg1 := THIS^.AnyToArg(currentValueAsString),
	arg2 := THIS^.AnyToArg(greaterValueAsString)
);

THIS^.assertorContainer.assertor.assert.dateAndTime.long.dateAndTime.valueIsLessThan(
	currentValue	:= valueToTest,
	greaterValue	:= greaterValue,
	message			:= ''
);

THIS^.AssertEquals_BOOL(
	Expected 	:= assertionIsWrong,
	Actual 		:= THIS^.assertorContainer.wasAssertionWrong,
	Message 	:= messageStringBuilder.sOut
);
END_METHOD

(*

short summary
==================
This test method tests ``assert.dateAndTime.long.dateAndTime.valueIsMax``
method of CNM_AssertionInterfaces library, 
it provides the possibility to handover test data via parameter 


.. <legal notes>

legal notes
=================
| SPDX-FileCopyrightText: © 2022 ekvip automation GmbH <info@ekvip.de>
| SPDX-License-Identifier: Apache-2.0
| For details check: Apache-2.0_

.. _Apache-2.0: https://www.apache.org/licenses/LICENSE-2.0

.. </legal notes>

parameters
==========

*)

METHOD testValueIsMax 
VAR_INPUT
	(* for the test it's the parameter ``currentValue`` *)
	valueToTest		:LDT;
	(* for the test it's the parameter ``greaterValue`` *)
	maximumValue	:LDT;
END_VAR
VAR
	(* just the expectation if the assertion to test must be worng or true *)
	assertionIsWrong		:BOOL;
	(* contains the format string for the test message *)
	message					:Tc2_System.T_MaxString;
	(* TwinCAT printf with the test message *)
	messageStringBuilder	:Tc2_Utilities.FB_FormatString;
	(* LDT value of ``currentValue`` as string *)
	currentValueAsString	:STRING(22);
	(* LDT value of ``maximumValue`` as string *)
	maximumValueAsString	:STRING(22);
END_VAR
THIS^.assertorContainer.resetAssertor();

assertionIsWrong := (valueToTest > maximumValue);

message := SEL(
	assertionIsWrong,
	'currentValue is %s maximumValue is %s assertion must be TRUE', 
	'currentValue is %s maximumValue is %s assertion must be FALSE'
);
currentValueAsString := TO_STRING(valueToTest);
maximumValueAsString := TO_STRING(maximumValue);

messageStringBuilder(
	sFormat := message,
	arg1 := THIS^.AnyToArg(currentValueAsString),
	arg2 := THIS^.AnyToArg(maximumValueAsString)
);

THIS^.assertorContainer.assertor.assert.dateAndTime.long.dateAndTime.valueIsMax(
	currentValue	:= valueToTest,
	maximumValue	:= maximumValue,
	message			:= ''
);

THIS^.AssertEquals_BOOL(
	Expected 	:= assertionIsWrong,
	Actual 		:= THIS^.assertorContainer.wasAssertionWrong,
	Message 	:= messageStringBuilder.sOut
);
END_METHOD

(*

short summary
==================
This test method tests ``assert.dateAndTime.long.dateAndTime.valueIsMin``
method of CNM_AssertionInterfaces library, 
it provides the possibility to handover test data via parameter 


.. <legal notes>

legal notes
=================
| SPDX-FileCopyrightText: © 2022 ekvip automation GmbH <info@ekvip.de>
| SPDX-License-Identifier: Apache-2.0
| For details check: Apache-2.0_

.. _Apache-2.0: https://www.apache.org/licenses/LICENSE-2.0

.. </legal notes>

parameters
==========

*)

METHOD testValueIsMin 
VAR_INPUT
	(* for the test it's the parameter ``currentValue`` *)
	valueToTest		:LDT;
	(* for the test it's the parameter ``greaterValue`` *)
	minimumValue	:LDT;
END_VAR
VAR
	(* just the expectation if the assertion to test must be worng or true *)
	assertionIsWrong		:BOOL;
	(* contains the format string for the test message *)
	message					:Tc2_System.T_MaxString;
	(* TwinCAT printf with the test message *)
	messageStringBuilder	:Tc2_Utilities.FB_FormatString;
	(* LDT value of ``currentValue`` as string *)
	currentValueAsString	:STRING(22);
	(* LDT value of ``minimumValue`` as string *)
	minimumValueAsString	:STRING(22);
END_VAR
THIS^.assertorContainer.resetAssertor();

assertionIsWrong := (valueToTest < minimumValue);

message := SEL(
	assertionIsWrong,
	'currentValue is %s minimumValue is %s assertion must be TRUE', 
	'currentValue is %s minimumValue is %s assertion must be FALSE'
);
currentValueAsString := TO_STRING(valueToTest);
minimumValueAsString := TO_STRING(minimumValue);

messageStringBuilder(
	sFormat := message,
	arg1 := THIS^.AnyToArg(currentValueAsString),
	arg2 := THIS^.AnyToArg(minimumValueAsString)
);

THIS^.assertorContainer.assertor.assert.dateAndTime.long.dateAndTime.valueIsMin(
	currentValue	:= valueToTest,
	minimumValue	:= minimumValue,
	message			:= ''
);

THIS^.AssertEquals_BOOL(
	Expected 	:= assertionIsWrong,
	Actual 		:= THIS^.assertorContainer.wasAssertionWrong,
	Message 	:= messageStringBuilder.sOut
);
END_METHOD

(*

short summary
==================
This test method tests ``assert.dateAndTime.long.dateAndTime.valueIsNotEqualTo``
method of CNM_AssertionInterfaces library, 
it provides the possibility to handover test data via parameter 


.. <legal notes>

legal notes
=================
| SPDX-FileCopyrightText: © 2022 ekvip automation GmbH <info@ekvip.de>
| SPDX-License-Identifier: Apache-2.0
| For details check: Apache-2.0_

.. _Apache-2.0: https://www.apache.org/licenses/LICENSE-2.0

.. </legal notes>

parameters
==========

*)

METHOD testValueIsNotEqualTo 
VAR_INPUT
	(* for the test it's the parameter ``currentValue`` *)
	valueToTest		:LDT;
	(* for the test it's the parameter ``unexpectedValue`` *)
	unexpectedValue	:LDT;
END_VAR
VAR
	(* just the expectation if the assertion to test must be worng or true *)
	assertionIsWrong		:BOOL;
	(* contains the format string for the test message *)
	message					:Tc2_System.T_MaxString;
	(* TwinCAT printf with the test message *)
	messageStringBuilder	:Tc2_Utilities.FB_FormatString;
	(* LDT value of ``currentValue`` as string *)
	currentValueAsString	:STRING(22);
	(* LDT value of ``unexpectedValue`` as string *)
	unexpectedValueAsString	:STRING(22);
END_VAR
THIS^.assertorContainer.resetAssertor();

assertionIsWrong := (valueToTest = unexpectedValue);

message := SEL(
	assertionIsWrong,
	'currentValue is %s expectedValue is %s assertion must be TRUE', 
	'currentValue is %s expectedValue is %s assertion must be FALSE'
);
currentValueAsString := TO_STRING(valueToTest);
unexpectedValueAsString := TO_STRING(unexpectedValue);

messageStringBuilder(
	sFormat := message,
	arg1 := THIS^.AnyToArg(currentValueAsString),
	arg2 := THIS^.AnyToArg(unexpectedValueAsString)
);

THIS^.assertorContainer.assertor.assert.dateAndTime.long.dateAndTime.valueIsNotEqualTo(
	currentValue	:= valueToTest,
	unexpectedValue	:= unexpectedValue,
	message			:= ''
);

THIS^.AssertEquals_BOOL(
	Expected 	:= assertionIsWrong,
	Actual 		:= THIS^.assertorContainer.wasAssertionWrong,
	Message 	:= messageStringBuilder.sOut
);
END_METHOD

END_FUNCTION_BLOCK

// ---- AssertionTester/AssertionTests/DateTimeAssertions/classes/LTODAssertionTests.TcPOU
(*

short summary
==================
This class tests all methods of LTOD assertions
with various combinations of inputs and checks expected 
outputs are satisfied or not

.. <legal notes>

legal notes
=================
| SPDX-FileCopyrightText: © 2022 ekvip automation GmbH <info@ekvip.de>
| SPDX-License-Identifier: Apache-2.0
| For details check: Apache-2.0_

.. _Apache-2.0: https://www.apache.org/licenses/LICENSE-2.0

.. </legal notes>

methods and properties
======================

*)


FUNCTION_BLOCK LTODAssertionTests EXTENDS AbstractAssertorTest
VAR
	
END_VAR
VAR CONSTANT
	(* prefix to unify the test names *)
	TEST_NAME_PREFIX		:STRING := 'assert.dateAndTime.long.timeOfDay.';
	(* max value of a LWORD *)
	{attribute 'hide'}
	MAX_LWORD				:LWORD := 16#FFFF_FFFF_FFFF_FFFF;
	(* min value of a LWORD *)
	{attribute 'hide'}
	MIN_LWORD				:LWORD := 16#0000_0000_0000_0000;
	(* only the msb is set *)
	{attribute 'hide'}
	MSB_ONLY				:LWORD := 16#8000_0000_0000_0000;
	(* only the msb is set *)
	{attribute 'hide'}
	LSB_ONLY				:LWORD := 16#0000_0000_0000_0001;
	(* all bits set except the msb *)
	{attribute 'hide'}
	WITHOUT_MSB 			:LWORD := 16#7FFF_FFFF_FFFF_FFFF;
	(* for every nibble is the msb set only *)
	{attribute 'hide'}
	ALL_NIBBLE_MSB			:LWORD := 16#8888_8888_8888_8888;
	(* for every nibble is the msb unset only *)
	{attribute 'hide'}
	WITHOUT_NIBBLE_MSB		:LWORD := 16#7777_7777_7777_7777;
	(* for every nibble is the lsb set only *)
	{attribute 'hide'}
	ALL_NIBBLE_LSB			:LWORD := 16#1111_1111_1111_1111;
	(* every bit is set except the lsb *)
	{attribute 'hide'}
	LSB_IS_UNSET			:LWORD := 16#FFFF_FFFF_FFFF_FFFE;
	(* max vale of time of day *)
	LTOD_MAX				:LTOD := TO_LTOD(MAX_LWORD);
	(* min vale of time of day *)
	LTOD_MIN				:LTOD := TO_LTOD(MIN_LWORD);
	(* only the msb is set *)
	LTOD_MSB_ONLY			:LTOD := TO_LTOD(MSB_ONLY);
	(* all bits set except the msb *)
	LTOD_WITHOUT_MSB 		:LTOD := TO_LTOD(WITHOUT_MSB);
	(* for every nibble is the msb set only *)
	LTOD_ALL_NIBBLE_MSB		:LTOD := TO_LTOD(ALL_NIBBLE_MSB);
	(* for every nibble is the msb unset only *)
	LTOD_WITHOUT_NIBBLE_MSB	:LTOD := TO_LTOD(WITHOUT_NIBBLE_MSB);
	(* for every nibble is the lsb set only *)
	LTOD_ALL_NIBBLE_LSB		:LTOD := TO_LTOD(ALL_NIBBLE_LSB);	
	(* every bit is set except the lsb *)
	LTOD_LSB_IS_UNSET		:LTOD := TO_LTOD(LSB_IS_UNSET);
	(* only the msb is set *)
	LTOD_LSB_ONLY			:LTOD := TO_LTOD(LSB_ONLY);
END_VAR

THIS^.runValueIsEqualToTests();
THIS^.runValueIsGreaterThanTests();
THIS^.runValueIsInRangeOfTests();
THIS^.runValueIsLessThanTests();
THIS^.runValueIsMaxTests();
THIS^.runValueIsMinTests();
THIS^.runValueIsNotEqualToTests();

(*

short summary
==================
This test method is a helper function to create a unified test name

.. <legal notes>

legal notes
=================
| SPDX-FileCopyrightText: © 2022 ekvip automation GmbH <info@ekvip.de>
| SPDX-License-Identifier: Apache-2.0
| For details check: Apache-2.0_

.. _Apache-2.0: https://www.apache.org/licenses/LICENSE-2.0

.. </legal notes>

parameters
==========

*)

METHOD PROTECTED getTestNameFor :Tc2_System.T_MaxString
VAR_INPUT
	(* name of the method to test, to create a unified test name *)
	nameOfMethodToTest	:Tc2_System.T_MaxString;
END_VAR
getTestNameFor := Tc2_Standard.CONCAT(THIS^.TEST_NAME_PREFIX, nameOfMethodToTest);
END_METHOD

(*

short summary
==================
This test method tests ``assert.dateAndTime.long.timeOfDay.valueIsEqualTo``
method of CNM_AssertionInterfaces library with various inputs

.. <legal notes>

legal notes
=================
| SPDX-FileCopyrightText: © 2022 ekvip automation GmbH <info@ekvip.de>
| SPDX-License-Identifier: Apache-2.0
| For details check: Apache-2.0_

.. _Apache-2.0: https://www.apache.org/licenses/LICENSE-2.0

.. </legal notes>

*)

METHOD runValueIsEqualToTests
RETURN (NOT TcUnit.TEST_ORDERED(THIS^.getTestNameFor('valueIsEqualTo')));

THIS^.testValueIsEqualTo(
	valueToTest := THIS^.LTOD_MAX,
	expected := THIS^.LTOD_MAX
);
THIS^.testValueIsEqualTo(
	valueToTest := THIS^.LTOD_MIN,
	expected := THIS^.LTOD_MIN
);
THIS^.testValueIsEqualTo(
	valueToTest := THIS^.LTOD_MIN,
	expected := THIS^.LTOD_MAX
);
THIS^.testValueIsEqualTo(
	valueToTest := THIS^.LTOD_MAX,
	expected := THIS^.LTOD_MIN
);
THIS^.testValueIsEqualTo(
	valueToTest := THIS^.LTOD_ALL_NIBBLE_LSB,
	expected := THIS^.LTOD_ALL_NIBBLE_LSB
);
THIS^.testValueIsEqualTo(
	valueToTest := THIS^.LTOD_LSB_ONLY,
	expected := THIS^.LTOD_MSB_ONLY
);
THIS^.testValueIsEqualTo(
	valueToTest := THIS^.LTOD_MSB_ONLY,
	expected := THIS^.LTOD_MSB_ONLY
);
THIS^.testValueIsEqualTo(
	valueToTest := THIS^.LTOD_MSB_ONLY,
	expected := THIS^.LTOD_LSB_ONLY
);

TcUnit.TEST_FINISHED();
END_METHOD

(*

short summary
==================
This test method tests ``assert.dateAndTime.long.timeOfDay.valueIsGreaterThan``
method of CNM_AssertionInterfaces library with various inputs

.. <legal notes>

legal notes
=================
| SPDX-FileCopyrightText: © 2022 ekvip automation GmbH <info@ekvip.de>
| SPDX-License-Identifier: Apache-2.0
| For details check: Apache-2.0_

.. _Apache-2.0: https://www.apache.org/licenses/LICENSE-2.0

.. </legal notes>

*)

METHOD runValueIsGreaterThanTests
RETURN (NOT TcUnit.TEST_ORDERED(THIS^.getTestNameFor('valueIsGreaterThan')));

